RoboDK station: final_robot_station.rdk

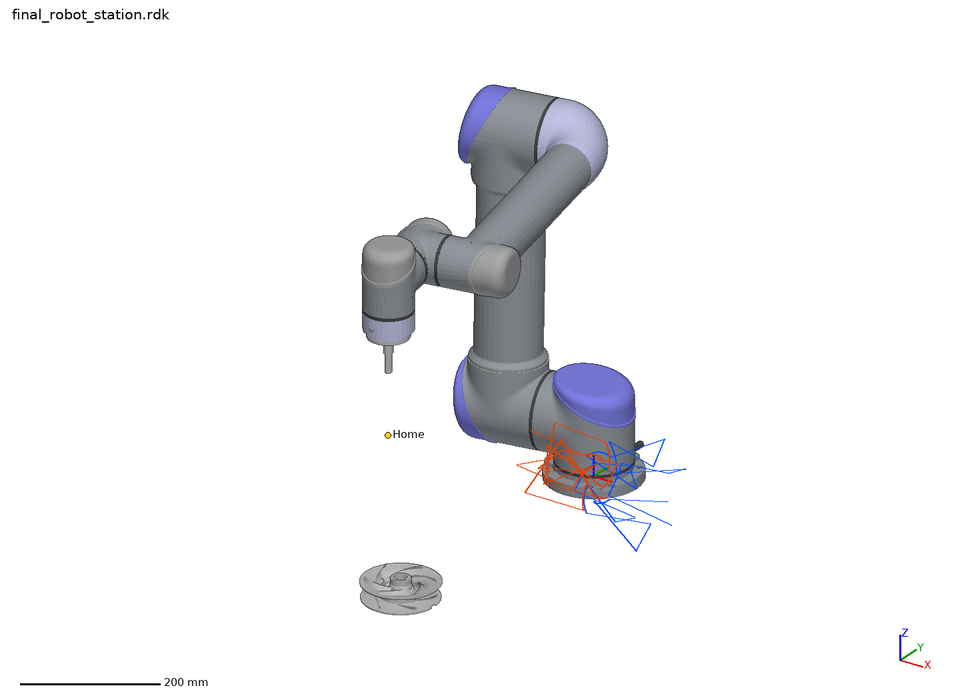
[picture v0: the station drawn from its stored meshes, robots at their saved joint values, targets as dots, program paths as lines]
Station test3. Poses are relative to the parent item; angles as X-Y-Z fixed-axis rotations.
  - frame UR5 Base at (0, 0, 0) mm, rotated rx 0 ry 0 rz -2.6 deg
    - robot UR5: 6 axes, payload 5 kg, reach 850 mm, repeatability 0.1 mm, weight 18.4 kg
        modified DH rows (alpha deg, a mm, theta deg, d mm): 0, 0, 0, 89.2; 90, 0, 180, 0; 0, 425, 0, 0; 0, 392.43, 0, 109; -90, 0, 0, 93.65; 90, 0, 180, 82
        joint limits [-360, -360, -360, -360, -360, -360] to [360, 360, 360, 360, 360, 360]; home [0, -90, -90, 0, 90, 0]; saved at [-76.875, -87.55, -95.198, -87.252, 90, 13.125]
      - tool laser_fixture_tool, TCP at (0, 0, 163) mm, size 63 x 63 x 63 mm
    - target Home (joint target) at (0, -480, 250) mm, rotated rx -180 ry 0 rz -180 deg; joints [-76.875, -87.55, -95.198, -87.252, 90, 13.125] of UR5
  - machining project Path1 settings: rotZ(0) | rotX(0)*rotY(0) | rotz(0) | onStart | onPathStart | onApproach | onPoint | onRetract | onFinish | SetRPM(%1) | SetTool(%1) | Extruder(%1) | default | default | OutOnMov(%1) | OutOffMov(%1) | onPathFinish | M_RunCode(%1)
  - program upper_vane (336 instructions, listed below)
  - machining project Path2 settings: rotZ(0) | rotX(0)*rotY(0) | rotz(0) | onStart | onPathStart | onApproach | onPoint | onRetract | onFinish | SetRPM(%1) | SetTool(%1) | Extruder(%1) | default | default | OutOnMov(%1) | OutOffMov(%1) | onPathFinish | M_RunCode(%1)
  - program lower_vane (305 instructions, listed below)
  - machining project Path3 settings: rotZ(0) | rotX(0)*rotY(0) | rotz(0) | onStart | onPathStart | onApproach | onPoint | onRetract | onFinish | SetRPM(%1) | SetTool(%1) | Extruder(%1) | default | default | OutOnMov(%1) | OutOffMov(%1) | onPathFinish | M_RunCode(%1)
  - program hub (106 instructions, listed below)
  - object PAPER_TEST at (0, -480, 0) mm, size 98 x 86 x 16 mm, geometry from PAPER_TEST.step
  - program MainProgram (19 instructions, listed below)
  - program Path2 (299 instructions, listed below)
  - program Path3 (105 instructions, listed below)
  - frame table at (0, 0, 0) mm
  - object Top_weld_path_dense at (0, -480, 0) mm, rotated rx 0 ry -90 rz 0 deg, size 32.2 x 115.4 x 114.9 mm
  - object Lower_weld_path_dense at (0, 0, 32.2) mm, rotated rx 0 ry 90 rz 0 deg, size 31 x 118.2 x 118.2 mm
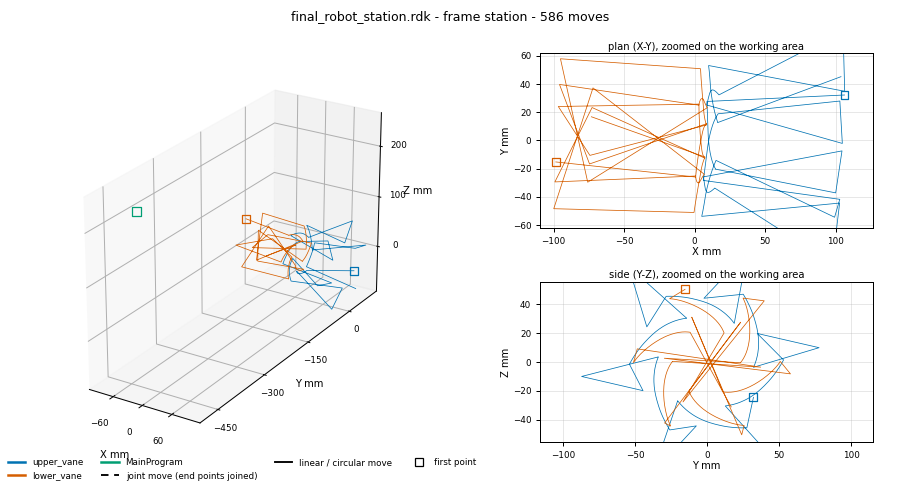
[picture p0: tool path of final_robot_station.rdk in frame station, 586 of 1059 moves have a stored position in this frame; points joined in program order, loops and branches not executed]
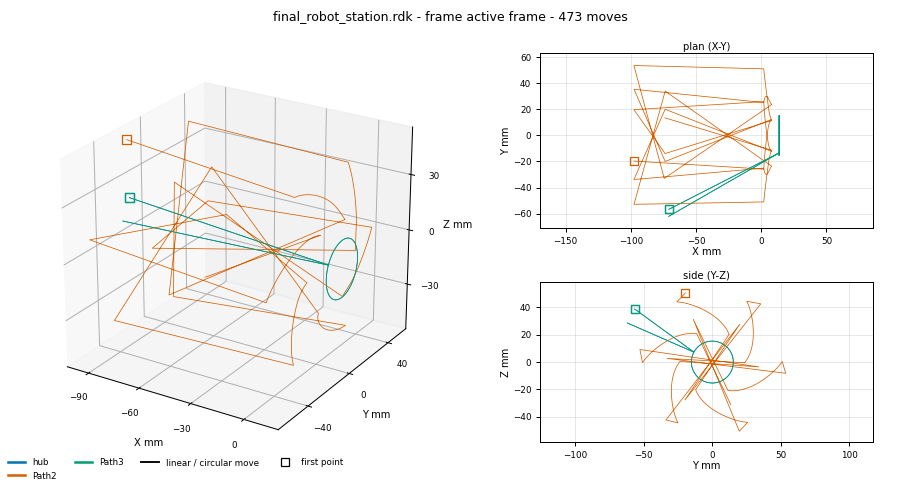
[picture p1: tool path of final_robot_station.rdk in frame active frame, 473 of 1059 moves have a stored position in this frame; points joined in program order, loops and branches not executed]

--- program upper_vane (robot UR5) ---
  Smooth(1)
  Set Ref.: UR5 Base
  Set Tool: laser_fixture_tool
  Show laser_fixture_tool
  Set speed (1000.0 mm/s)
  MoveJ 1 to (104.83, 37.05, -24.45) mm, rotated rx -180 ry -77.76 rz -174.71 deg; joints [-78.761, -85.544, -122.094, -54.774, 100.978, 11.402]
  MoveL 2 to (104.83, 37.05, -24.45) mm, rotated rx -180 ry -77.76 rz -174.71 deg; joints [-78.761, -85.544, -122.094, -54.774, 100.978, 11.402]
  MoveL 3 to (7.52, 28.05, -45.66) mm, rotated rx 180 ry -77.76 rz -174.71 deg; joints [-76.153, -96.353, -128.923, -36.642, 100.622, 14.033]
  MoveL 4 to (7.52, 28.05, -45.66) mm, rotated rx 180 ry -77.76 rz -174.71 deg; joints [-76.153, -96.353, -128.923, -36.642, 100.622, 14.033]
  Set speed (100.0 mm/s)
  Smooth(1)
  MoveL 5 to (7.65, 26.53, -45.69) mm, rotated rx 180 ry -78.61 rz -174.54 deg; joints [-75.694, -96.347, -128.777, -36.756, 99.685, 14.45]
  MoveL 6 to (7.78, 25.01, -45.69) mm, rotated rx -180 ry -79.74 rz -174.38 deg; joints [-75.091, -96.317, -128.596, -37.013, 98.472, 15.003]
  MoveL 7 to (7.91, 23.49, -45.67) mm, rotated rx 180 ry -81.09 rz -174.3 deg; joints [-74.379, -96.291, -128.35, -37.468, 97.046, 15.663]
  MoveL 8 to (8.03, 22.04, -45.61) mm, rotated rx 180 ry -82.56 rz -174.26 deg; joints [-73.616, -96.281, -128.06, -38.061, 95.524, 16.378]
  MoveL 9 to (8.15, 20.65, -45.54) mm, rotated rx 180 ry -84.09 rz -174.26 deg; joints [-72.832, -96.291, -127.75, -38.731, 93.961, 17.121]
  MoveL 10 to (8.26, 19.26, -45.44) mm, rotated rx 180 ry -85.7 rz -174.3 deg; joints [-72.021, -96.337, -127.386, -39.533, 92.34, 17.903]
  MoveL 11 to (8.37, 17.87, -45.32) mm, rotated rx 180 ry -87.36 rz -174.38 deg; joints [-71.197, -96.422, -126.982, -40.43, 90.689, 18.711]
  MoveL 12 to (8.49, 16.49, -45.17) mm, rotated rx 180 ry -89.06 rz -174.48 deg; joints [-70.375, -96.543, -126.553, -41.387, 89.033, 19.533]
  MoveL 13 to (8.6, 15.11, -44.99) mm, rotated rx 0 ry -89.24 rz 5.33 deg; joints [-69.589, -96.729, -126.039, -42.503, 87.434, 20.341]
  MoveL 14 to (8.7, 13.77, -44.79) mm, rotated rx 0 ry -87.62 rz 4.97 deg; joints [-68.892, -96.992, -125.413, -43.811, 85.994, 21.079]
  MoveL 15 to (8.8, 12.48, -44.57) mm, rotated rx 0 ry -86.09 rz 4.54 deg; joints [-68.268, -97.304, -124.741, -45.182, 84.684, 21.758]
  MoveL 16 to (8.9, 11.19, -44.33) mm, rotated rx 0 ry -84.61 rz 3.98 deg; joints [-67.718, -97.686, -123.97, -46.708, 83.499, 22.377]
  MoveL 17 to (9, 9.83, -44.04) mm, rotated rx 0 ry -83.06 rz 3.41 deg; joints [-67.162, -98.115, -123.162, -48.289, 82.283, 23.016]
  MoveL 18 to (9.1, 8.47, -43.73) mm, rotated rx 0 ry -81.52 rz 2.91 deg; joints [-66.609, -98.544, -122.405, -49.771, 81.062, 23.664]
  MoveL 19 to (9.21, 7.11, -43.4) mm, rotated rx 0 ry -79.92 rz 2.67 deg; joints [-65.995, -98.917, -121.82, -50.973, 79.719, 24.393]
  MoveL 20 to (9.32, 5.84, -43.07) mm, rotated rx 0 ry -78.4 rz 2.53 deg; joints [-65.401, -99.258, -121.333, -52.005, 78.412, 25.12]
  MoveL 21 to (9.44, 4.58, -42.73) mm, rotated rx 0 ry -76.9 rz 2.35 deg; joints [-64.845, -99.631, -120.812, -53.094, 77.169, 25.822]
  MoveL 22 to (9.56, 3.42, -42.39) mm, rotated rx 0 ry -75.57 rz 2.15 deg; joints [-64.375, -99.996, -120.31, -54.126, 76.093, 26.437]
  MoveL 23 to (9.67, 2.38, -42.07) mm, rotated rx 0 ry -74.39 rz 2 deg; joints [-63.962, -100.325, -119.878, -55.019, 75.134, 26.993]
  MoveL 24 to (9.79, 1.35, -41.73) mm, rotated rx 0 ry -73.25 rz 1.82 deg; joints [-63.588, -100.667, -119.429, -55.928, 74.241, 27.514]
  MoveL 25 to (9.91, 0.35, -41.38) mm, rotated rx 0 ry -72.21 rz 1.6 deg; joints [-63.268, -101.011, -118.973, -56.827, 73.449, 27.974]
  MoveL 26 to (10.04, -0.61, -41.02) mm, rotated rx 0 ry -71.25 rz 1.39 deg; joints [-62.988, -101.342, -118.538, -57.674, 72.731, 28.39]
  MoveL 27 to (10.18, -1.55, -40.65) mm, rotated rx 0 ry -70.36 rz 1.15 deg; joints [-62.753, -101.677, -118.092, -58.517, 72.092, 28.754]
  MoveL 28 to (10.33, -2.51, -40.24) mm, rotated rx 0 ry -69.54 rz 0.86 deg; joints [-62.564, -102.018, -117.626, -59.366, 71.534, 29.06]
  MoveL 29 to (10.48, -3.45, -39.82) mm, rotated rx 0 ry -68.79 rz 0.57 deg; joints [-62.41, -102.352, -117.166, -60.183, 71.038, 29.32]
  MoveL 30 to (10.65, -4.38, -39.38) mm, rotated rx 0 ry -68.11 rz 0.26 deg; joints [-62.291, -102.677, -116.711, -60.968, 70.604, 29.534]
  MoveL 31 to (10.82, -5.3, -38.92) mm, rotated rx 0 ry -67.47 rz 0 deg; joints [-62.186, -102.982, -116.291, -61.687, 70.191, 29.733]
  MoveL 32 to (11.01, -6.25, -38.41) mm, rotated rx 0 ry -66.89 rz -0.34 deg; joints [-62.125, -103.301, -115.833, -62.437, 69.851, 29.869]
  MoveL 33 to (11.21, -7.19, -37.88) mm, rotated rx 0 ry -66.37 rz -0.67 deg; joints [-62.092, -103.605, -115.389, -63.143, 69.562, 29.964]
  MoveL 34 to (11.42, -8.11, -37.33) mm, rotated rx 0 ry -65.93 rz -1.01 deg; joints [-62.095, -103.898, -114.948, -63.819, 69.339, 30.006]
  MoveL 35 to (11.64, -9.02, -36.76) mm, rotated rx 0 ry -65.54 rz -1.35 deg; joints [-62.117, -104.173, -114.529, -64.444, 69.148, 30.021]
  MoveL 36 to (11.86, -9.91, -36.17) mm, rotated rx 0 ry -65.18 rz -1.65 deg; joints [-62.144, -104.43, -114.137, -65.021, 68.967, 30.026]
  MoveL 37 to (12.1, -10.79, -35.56) mm, rotated rx 0 ry -64.87 rz -1.99 deg; joints [-62.198, -104.685, -113.735, -65.598, 68.834, 29.991]
  MoveL 38 to (12.33, -11.6, -34.96) mm, rotated rx 0 ry -64.54 rz -2.25 deg; joints [-62.224, -104.908, -113.396, -66.098, 68.659, 29.996]
  MoveL 39 to (12.58, -12.39, -34.35) mm, rotated rx 0 ry -64.18 rz -2.48 deg; joints [-62.236, -105.126, -113.072, -66.587, 68.454, 30.023]
  MoveL 40 to (12.84, -13.19, -33.7) mm, rotated rx 0 ry -63.8 rz -2.73 deg; joints [-62.245, -105.354, -112.733, -67.11, 68.233, 30.058]
  MoveL 41 to (13.12, -13.99, -33.01) mm, rotated rx 0 ry -63.4 rz -3.03 deg; joints [-62.261, -105.602, -112.358, -67.695, 68.019, 30.081]
  MoveL 42 to (13.41, -14.77, -32.31) mm, rotated rx 0 ry -62.99 rz -3.38 deg; joints [-62.285, -105.87, -111.95, -68.339, 67.816, 30.092]
  MoveL 43 to (13.7, -15.51, -31.61) mm, rotated rx 0 ry -62.56 rz -3.76 deg; joints [-62.303, -106.15, -111.524, -69.027, 67.609, 30.107]
  MoveL 44 to (14, -16.21, -30.91) mm, rotated rx 0 ry -62.09 rz -4.16 deg; joints [-62.306, -106.443, -111.086, -69.759, 67.376, 30.144]
  MoveL 45 to (14.31, -16.89, -30.2) mm, rotated rx 0 ry -61.58 rz -4.62 deg; joints [-62.308, -106.766, -110.604, -70.575, 67.142, 30.178]
  MoveL 46 to (14.63, -17.55, -29.48) mm, rotated rx 0 ry -61.04 rz -5.16 deg; joints [-62.313, -107.122, -110.072, -71.483, 66.91, 30.203]
  MoveL 47 to (14.97, -18.18, -28.74) mm, rotated rx 0 ry -60.48 rz -5.78 deg; joints [-62.325, -107.517, -109.481, -72.493, 66.694, 30.208]
  MoveL 48 to (15.31, -18.8, -28) mm, rotated rx 0 ry -59.9 rz -6.49 deg; joints [-62.345, -107.949, -108.834, -73.6, 66.494, 30.193]
  MoveL 49 to (15.66, -19.38, -27.25) mm, rotated rx 0 ry -59.71 rz -7.57 deg; joints [-62.575, -108.441, -107.984, -74.851, 66.721, 29.804]
  MoveL 50 to (15.84, -19.66, -26.87) mm, rotated rx 0 ry -60.27 rz -8.58 deg; joints [-63.004, -108.736, -107.315, -75.582, 67.472, 29.074]
  Set speed (1000.0 mm/s)
  MoveL 51 to (15.84, -19.66, -26.87) mm, rotated rx 0 ry -60.27 rz -8.58 deg; joints [-63.004, -108.736, -107.315, -75.582, 67.472, 29.074]
  MoveL 52 to (101.71, -32.61, -76.47) mm, rotated rx 0 ry -60.27 rz -8.58 deg; joints [-59.167, -106.315, -95.895, -90.843, 68.931, 32.896]
  Set speed (1000.0 mm/s)
  MoveL 53 to (104.83, -2.65, -44.31) mm, rotated rx 180 ry -88.39 rz -166.78 deg; joints [-70.24, -87.361, -121.86, -47.778, 87.082, 19.241]
  MoveL 54 to (7.52, -25.52, -47.12) mm, rotated rx -180 ry -88.39 rz -166.78 deg; joints [-70.907, -100.111, -125.994, -30.862, 87.233, 18.59]
  MoveL 55 to (7.52, -25.52, -47.12) mm, rotated rx -180 ry -88.39 rz -166.78 deg; joints [-70.907, -100.111, -125.994, -30.862, 87.233, 18.59]
  Set speed (100.0 mm/s)
  Smooth(1)
  MoveL 56 to (7.65, -26.3, -45.82) mm, rotated rx -180 ry -88.98 rz -167.43 deg; joints [-70.908, -100.255, -125.373, -32.142, 86.887, 18.646]
  MoveL 57 to (7.78, -27.07, -44.51) mm, rotated rx -180 ry -89.68 rz -168.32 deg; joints [-70.892, -100.451, -124.564, -33.83, 86.506, 18.733]
  MoveL 58 to (7.91, -27.8, -43.18) mm, rotated rx 0 ry -89.56 rz 10.56 deg; joints [-70.888, -100.712, -123.582, -35.862, 86.148, 18.82]
  MoveL 59 to (8.03, -28.48, -41.89) mm, rotated rx 0 ry -88.79 rz 9.31 deg; joints [-70.894, -101.028, -122.505, -38.056, 85.822, 18.897]
  MoveL 60 to (8.15, -29.11, -40.65) mm, rotated rx 0 ry -88.01 rz 8 deg; joints [-70.9, -101.391, -121.379, -40.316, 85.512, 18.967]
  MoveL 61 to (8.26, -29.72, -39.4) mm, rotated rx 0 ry -87.24 rz 6.58 deg; joints [-70.926, -101.815, -120.171, -42.69, 85.24, 19.011]
  MoveL 62 to (8.37, -30.31, -38.14) mm, rotated rx 0 ry -86.46 rz 5.1 deg; joints [-70.965, -102.296, -118.908, -45.126, 84.994, 19.032]
  MoveL 63 to (8.49, -30.87, -36.86) mm, rotated rx 0 ry -85.69 rz 3.58 deg; joints [-71.011, -102.824, -117.611, -47.582, 84.761, 19.033]
  MoveL 64 to (8.6, -31.41, -35.58) mm, rotated rx 0 ry -85.01 rz 2.01 deg; joints [-71.107, -103.402, -116.278, -50.039, 84.629, 18.968]
  MoveL 65 to (8.7, -31.91, -34.32) mm, rotated rx 0 ry -84.51 rz 0.42 deg; joints [-71.28, -104.01, -114.951, -52.406, 84.664, 18.804]
  MoveL 66 to (8.8, -32.36, -33.09) mm, rotated rx 0 ry -84.11 rz -1.13 deg; joints [-71.487, -104.628, -113.66, -54.655, 84.776, 18.59]
  MoveL 67 to (8.9, -32.79, -31.86) mm, rotated rx 0 ry -83.86 rz -2.7 deg; joints [-71.756, -105.274, -112.363, -56.851, 85.016, 18.295]
  MoveL 68 to (9, -33.23, -30.53) mm, rotated rx 0 ry -83.59 rz -4.33 deg; joints [-72.028, -105.971, -111.011, -59.116, 85.243, 17.983]
  MoveL 69 to (9.1, -33.64, -29.2) mm, rotated rx 0 ry -83.26 rz -5.93 deg; joints [-72.258, -106.68, -109.682, -61.334, 85.386, 17.703]
  MoveL 70 to (9.21, -34.03, -27.86) mm, rotated rx 0 ry -82.7 rz -7.45 deg; joints [-72.369, -107.39, -108.393, -63.52, 85.284, 17.539]
  MoveL 71 to (9.32, -34.38, -26.6) mm, rotated rx 0 ry -82.07 rz -8.86 deg; joints [-72.426, -108.072, -107.192, -65.559, 85.093, 17.423]
  MoveL 72 to (9.44, -34.72, -25.33) mm, rotated rx 0 ry -81.5 rz -10.27 deg; joints [-72.505, -108.765, -105.998, -67.558, 84.947, 17.275]
  MoveL 73 to (9.56, -35, -24.16) mm, rotated rx 0 ry -81.02 rz -11.54 deg; joints [-72.595, -109.402, -104.922, -69.337, 84.849, 17.114]
  MoveL 74 to (9.67, -35.24, -23.1) mm, rotated rx 0 ry -80.58 rz -12.66 deg; joints [-72.664, -109.975, -103.972, -70.904, 84.735, 16.975]
  MoveL 75 to (9.79, -35.46, -22.03) mm, rotated rx 0 ry -80.19 rz -13.76 deg; joints [-72.748, -110.537, -103.051, -72.407, 84.652, 16.818]
  MoveL 76 to (9.91, -35.66, -21) mm, rotated rx 0 ry -79.87 rz -14.79 deg; joints [-72.849, -111.068, -102.191, -73.796, 84.612, 16.642]
  MoveL 77 to (10.04, -35.83, -19.99) mm, rotated rx 0 ry -79.59 rz -15.75 deg; joints [-72.95, -111.563, -101.397, -75.073, 84.581, 16.468]
  MoveL 78 to (10.18, -35.98, -18.98) mm, rotated rx 0 ry -79.37 rz -16.65 deg; joints [-73.067, -112.032, -100.648, -76.264, 84.584, 16.277]
  MoveL 79 to (10.33, -36.1, -17.95) mm, rotated rx 0 ry -79.22 rz -17.52 deg; joints [-73.206, -112.475, -99.941, -77.374, 84.629, 16.066]
  MoveL 80 to (10.48, -36.21, -16.92) mm, rotated rx 0 ry -79.11 rz -18.32 deg; joints [-73.352, -112.887, -99.286, -78.399, 84.689, 15.851]
  MoveL 81 to (10.65, -36.29, -15.9) mm, rotated rx 0 ry -79.04 rz -19.07 deg; joints [-73.505, -113.268, -98.68, -79.34, 84.765, 15.633]
  MoveL 82 to (10.82, -36.35, -14.87) mm, rotated rx 0 ry -78.96 rz -19.76 deg; joints [-73.646, -113.621, -98.121, -80.216, 84.818, 15.431]
  MoveL 83 to (11.01, -36.39, -13.79) mm, rotated rx 0 ry -78.95 rz -20.43 deg; joints [-73.816, -113.954, -97.588, -81.037, 84.922, 15.201]
  MoveL 84 to (11.21, -36.4, -12.71) mm, rotated rx 0 ry -78.98 rz -21.04 deg; joints [-73.99, -114.253, -97.108, -81.777, 85.035, 14.974]
  MoveL 85 to (11.42, -36.39, -11.64) mm, rotated rx 0 ry -79.05 rz -21.59 deg; joints [-74.174, -114.516, -96.681, -82.431, 85.17, 14.743]
  MoveL 86 to (11.64, -36.35, -10.57) mm, rotated rx 0 ry -79.14 rz -22.09 deg; joints [-74.355, -114.747, -96.3, -83.018, 85.301, 14.521]
  MoveL 87 to (11.86, -36.28, -9.5) mm, rotated rx 0 ry -79.21 rz -22.55 deg; joints [-74.526, -114.958, -95.951, -83.564, 85.414, 14.312]
  MoveL 88 to (12.1, -36.19, -8.44) mm, rotated rx 0 ry -79.33 rz -22.97 deg; joints [-74.71, -115.147, -95.632, -84.06, 85.556, 14.095]
  MoveL 89 to (12.33, -36.07, -7.44) mm, rotated rx 0 ry -79.38 rz -23.38 deg; joints [-74.857, -115.328, -95.329, -84.549, 85.639, 13.914]
  MoveL 90 to (12.58, -35.94, -6.44) mm, rotated rx 0 ry -79.4 rz -23.8 deg; joints [-74.992, -115.517, -95.017, -85.06, 85.697, 13.745]
  MoveL 91 to (12.84, -35.78, -5.43) mm, rotated rx 0 ry -79.41 rz -24.25 deg; joints [-75.129, -115.719, -94.686, -85.609, 85.758, 13.57]
  MoveL 92 to (13.12, -35.58, -4.39) mm, rotated rx 0 ry -79.46 rz -24.74 deg; joints [-75.282, -115.935, -94.331, -86.192, 85.846, 13.377]
  MoveL 93 to (13.41, -35.36, -3.36) mm, rotated rx 0 ry -79.54 rz -25.25 deg; joints [-75.449, -116.165, -93.956, -86.804, 85.967, 13.168]
  MoveL 94 to (13.7, -35.13, -2.37) mm, rotated rx 0 ry -79.63 rz -25.8 deg; joints [-75.617, -116.412, -93.558, -87.45, 86.101, 12.953]
  MoveL 95 to (14, -34.88, -1.42) mm, rotated rx 0 ry -79.72 rz -26.4 deg; joints [-75.783, -116.685, -93.124, -88.153, 86.237, 12.737]
  MoveL 96 to (14.31, -34.6, -0.47) mm, rotated rx 0 ry -79.83 rz -27.05 deg; joints [-75.962, -116.989, -92.649, -88.915, 86.404, 12.502]
  MoveL 97 to (14.63, -34.3, 0.46) mm, rotated rx 0 ry -79.98 rz -27.76 deg; joints [-76.157, -117.324, -92.13, -89.74, 86.607, 12.246]
  MoveL 98 to (14.97, -33.98, 1.38) mm, rotated rx 0 ry -80.19 rz -28.52 deg; joints [-76.373, -117.689, -91.568, -90.622, 86.858, 11.965]
  MoveL 99 to (15.31, -33.64, 2.28) mm, rotated rx 0 ry -80.44 rz -29.34 deg; joints [-76.61, -118.086, -90.964, -91.559, 87.154, 11.661]
  MoveL 100 to (15.66, -33.29, 3.16) mm, rotated rx 0 ry -81.17 rz -29.97 deg; joints [-77.008, -118.36, -90.513, -92.187, 87.784, 11.239]
  MoveL 101 to (15.84, -33.1, 3.59) mm, rotated rx 0 ry -82.19 rz -29.93 deg; joints [-77.434, -118.27, -90.576, -91.96, 88.565, 10.872]
  Set speed (1000.0 mm/s)
  MoveL 102 to (15.84, -33.1, 3.59) mm, rotated rx 0 ry -82.19 rz -29.93 deg; joints [-77.434, -118.27, -90.576, -91.96, 88.565, 10.872]
  MoveL 103 to (101.71, -82.53, -9.99) mm, rotated rx 0 ry -82.19 rz -29.93 deg; joints [-77.222, -120.426, -73.678, -106.707, 88.674, 11.054]
  Set speed (1000.0 mm/s)
  MoveL 104 to (104.83, -39.7, -19.86) mm, rotated rx 0 ry -79.4 rz 8.11 deg; joints [-69.534, -94.529, -112.106, -59.512, 77.242, 20.788]
  MoveL 105 to (7.52, -53.56, -1.46) mm, rotated rx 0 ry -79.4 rz 8.11 deg; joints [-72.132, -104.254, -117.716, -43.595, 77.429, 18.133]
  MoveL 106 to (7.52, -53.56, -1.46) mm, rotated rx 0 ry -79.4 rz 8.11 deg; joints [-72.132, -104.254, -117.716, -43.595, 77.429, 18.133]
  Set speed (100.0 mm/s)
  Smooth(1)
  MoveL 107 to (7.65, -52.83, -0.13) mm, rotated rx 0 ry -79.66 rz 7.26 deg; joints [-72.499, -104.351, -117.217, -44.647, 77.958, 17.76]
  MoveL 108 to (7.78, -52.08, 1.19) mm, rotated rx 0 ry -80.07 rz 6.18 deg; joints [-72.964, -104.514, -116.551, -45.96, 78.697, 17.279]
  MoveL 109 to (7.91, -51.29, 2.49) mm, rotated rx 0 ry -80.65 rz 4.94 deg; joints [-73.523, -104.733, -115.763, -47.441, 79.637, 16.694]
  MoveL 110 to (8.03, -50.52, 3.72) mm, rotated rx 0 ry -81.34 rz 3.63 deg; joints [-74.127, -104.996, -114.914, -48.986, 80.68, 16.058]
  MoveL 111 to (8.15, -49.76, 4.89) mm, rotated rx 0 ry -82.08 rz 2.28 deg; joints [-74.746, -105.3, -114.026, -50.568, 81.764, 15.405]
  MoveL 112 to (8.26, -48.98, 6.04) mm, rotated rx 0 ry -82.92 rz 0.89 deg; joints [-75.4, -105.642, -113.098, -52.188, 82.924, 14.712]
  MoveL 113 to (8.37, -48.18, 7.18) mm, rotated rx 0 ry -83.82 rz -0.52 deg; joints [-76.075, -106.021, -112.143, -53.836, 84.125, 14]
  MoveL 114 to (8.49, -47.36, 8.3) mm, rotated rx 0 ry -84.75 rz -1.95 deg; joints [-76.753, -106.433, -111.169, -55.502, 85.336, 13.284]
  MoveL 115 to (8.6, -46.52, 9.41) mm, rotated rx 0 ry -85.77 rz -3.33 deg; joints [-77.454, -106.851, -110.233, -57.081, 86.594, 12.547]
  MoveL 116 to (8.7, -45.68, 10.47) mm, rotated rx 0 ry -86.89 rz -4.55 deg; joints [-78.169, -107.237, -109.409, -58.442, 87.889, 11.802]
  MoveL 117 to (8.8, -44.84, 11.48) mm, rotated rx 0 ry -88.03 rz -5.66 deg; joints [-78.868, -107.604, -108.665, -59.666, 89.16, 11.078]
  MoveL 118 to (8.9, -43.98, 12.47) mm, rotated rx 0 ry -89.26 rz -6.66 deg; joints [-79.587, -107.944, -108.008, -60.734, 90.474, 10.342]
  MoveL 119 to (9, -43.06, 13.51) mm, rotated rx 180 ry -89.47 rz 172.29 deg; joints [-80.323, -108.318, -107.317, -61.878, 91.816, 9.593]
  MoveL 120 to (9.1, -42.11, 14.53) mm, rotated rx 180 ry -88.27 rz 171.2 deg; joints [-81.021, -108.726, -106.593, -63.107, 93.079, 8.885]
  MoveL 121 to (9.21, -41.14, 15.54) mm, rotated rx 180 ry -87.26 rz 169.94 deg; joints [-81.635, -109.218, -105.728, -64.612, 94.169, 8.257]
  MoveL 122 to (9.32, -40.22, 16.48) mm, rotated rx 180 ry -86.38 rz 168.69 deg; joints [-82.175, -109.727, -104.856, -66.144, 95.115, 7.703]
  MoveL 123 to (9.44, -39.29, 17.4) mm, rotated rx -180 ry -85.49 rz 167.47 deg; joints [-82.71, -110.229, -104.021, -67.616, 96.055, 7.156]
  MoveL 124 to (9.56, -38.42, 18.23) mm, rotated rx 180 ry -84.66 rz 166.41 deg; joints [-83.192, -110.678, -103.295, -68.904, 96.903, 6.665]
  MoveL 125 to (9.67, -37.62, 18.97) mm, rotated rx 180 ry -83.95 rz 165.45 deg; joints [-83.606, -111.09, -102.638, -70.081, 97.623, 6.244]
  MoveL 126 to (9.79, -36.81, 19.7) mm, rotated rx 180 ry -83.24 rz 164.54 deg; joints [-84.009, -111.481, -102.027, -71.187, 98.325, 5.835]
  MoveL 127 to (9.91, -36.01, 20.38) mm, rotated rx 180 ry -82.55 rz 163.72 deg; joints [-84.392, -111.833, -101.49, -72.175, 98.991, 5.45]
  MoveL 128 to (10.04, -35.22, 21.04) mm, rotated rx 180 ry -81.9 rz 162.97 deg; joints [-84.745, -112.155, -101.006, -73.082, 99.602, 5.095]
  MoveL 129 to (10.18, -34.42, 21.67) mm, rotated rx 180 ry -81.27 rz 162.3 deg; joints [-85.086, -112.441, -100.585, -73.894, 100.19, 4.756]
  MoveL 130 to (10.33, -33.6, 22.29) mm, rotated rx 180 ry -80.64 rz 161.7 deg; joints [-85.419, -112.688, -100.231, -74.605, 100.765, 4.427]
  MoveL 131 to (10.48, -32.76, 22.9) mm, rotated rx 180 ry -80.05 rz 161.17 deg; joints [-85.735, -112.903, -99.93, -75.241, 101.305, 4.117]
  MoveL 132 to (10.65, -31.91, 23.48) mm, rotated rx -180 ry -79.47 rz 160.69 deg; joints [-86.034, -113.085, -99.679, -75.801, 101.815, 3.824]
  MoveL 133 to (10.82, -31.05, 24.05) mm, rotated rx -180 ry -78.95 rz 160.24 deg; joints [-86.308, -113.253, -99.448, -76.34, 102.277, 3.556]
  MoveL 134 to (11.01, -30.14, 24.62) mm, rotated rx 180 ry -78.41 rz 159.86 deg; joints [-86.588, -113.378, -99.285, -76.782, 102.747, 3.285]
  MoveL 135 to (11.21, -29.21, 25.17) mm, rotated rx -180 ry -77.9 rz 159.54 deg; joints [-86.849, -113.471, -99.17, -77.154, 103.185, 3.032]
  MoveL 136 to (11.42, -28.27, 25.69) mm, rotated rx 180 ry -77.41 rz 159.29 deg; joints [-87.097, -113.525, -99.113, -77.437, 103.598, 2.793]
  MoveL 137 to (11.64, -27.32, 26.19) mm, rotated rx -180 ry -76.97 rz 159.08 deg; joints [-87.327, -113.555, -99.089, -77.675, 103.976, 2.573]
  MoveL 138 to (11.86, -26.37, 26.67) mm, rotated rx 180 ry -76.55 rz 158.88 deg; joints [-87.539, -113.575, -99.075, -77.902, 104.324, 2.369]
  MoveL 139 to (12.1, -25.4, 27.12) mm, rotated rx 180 ry -76.14 rz 158.73 deg; joints [-87.748, -113.565, -99.105, -78.061, 104.668, 2.17]
  MoveL 140 to (12.33, -24.48, 27.52) mm, rotated rx 180 ry -75.78 rz 158.54 deg; joints [-87.93, -113.582, -99.091, -78.285, 104.967, 1.994]
  MoveL 141 to (12.58, -23.55, 27.9) mm, rotated rx -180 ry -75.43 rz 158.31 deg; joints [-88.107, -113.614, -99.051, -78.556, 105.259, 1.823]
  MoveL 142 to (12.84, -22.59, 28.27) mm, rotated rx -180 ry -75.06 rz 158.06 deg; joints [-88.292, -113.654, -99, -78.852, 105.571, 1.645]
  MoveL 143 to (13.12, -21.59, 28.62) mm, rotated rx 180 ry -74.64 rz 157.81 deg; joints [-88.493, -113.692, -98.959, -79.143, 105.919, 1.451]
  MoveL 144 to (13.41, -20.59, 28.95) mm, rotated rx 180 ry -74.18 rz 157.58 deg; joints [-88.709, -113.729, -98.927, -79.423, 106.305, 1.243]
  MoveL 145 to (13.7, -19.62, 29.24) mm, rotated rx -180 ry -73.69 rz 157.33 deg; joints [-88.934, -113.778, -98.884, -79.718, 106.716, 1.027]
  MoveL 146 to (14, -18.66, 29.49) mm, rotated rx 180 ry -73.17 rz 157.04 deg; joints [-89.168, -113.852, -98.811, -80.059, 107.155, 0.802]
  MoveL 147 to (14.31, -17.71, 29.73) mm, rotated rx 180 ry -72.58 rz 156.75 deg; joints [-89.423, -113.937, -98.733, -80.416, 107.644, 0.556]
  MoveL 148 to (14.63, -16.76, 29.94) mm, rotated rx 180 ry -71.93 rz 156.44 deg; joints [-89.702, -114.034, -98.651, -80.783, 108.189, 0.288]
  MoveL 149 to (14.97, -15.8, 30.12) mm, rotated rx -180 ry -71.2 rz 156.14 deg; joints [-90.007, -114.136, -98.577, -81.146, 108.796, -0.006]
  MoveL 150 to (15.31, -14.85, 30.28) mm, rotated rx -180 ry -70.4 rz 155.85 deg; joints [-90.336, -114.245, -98.51, -81.505, 109.462, -0.326]
  MoveL 151 to (15.66, -13.91, 30.41) mm, rotated rx -180 ry -69.47 rz 156.07 deg; joints [-90.715, -114.109, -98.833, -81.229, 110.241, -0.697]
  MoveL 152 to (15.84, -13.44, 30.46) mm, rotated rx 180 ry -68.89 rz 156.98 deg; joints [-90.952, -113.656, -99.593, -80.102, 110.734, -0.937]
  Set speed (1000.0 mm/s)
  MoveL 153 to (15.84, -13.44, 30.46) mm, rotated rx 180 ry -68.89 rz 156.98 deg; joints [-90.952, -113.656, -99.593, -80.102, 110.734, -0.937]
  MoveL 154 to (101.71, -49.91, 66.48) mm, rotated rx -180 ry -68.89 rz 156.98 deg; joints [-94.194, -113.921, -84.944, -95.571, 109.42, -4.093]
  Set speed (1000.0 mm/s)
  MoveL 155 to (104.83, -37.05, 24.45) mm, rotated rx 0 ry -77.76 rz -5.29 deg; joints [-75.431, -100.004, -102.645, -75.565, 79.48, 14.759]
  MoveL 156 to (7.52, -28.05, 45.66) mm, rotated rx 0 ry -77.76 rz -5.29 deg; joints [-77.455, -105.732, -111.895, -60.21, 79.198, 12.72]
  MoveL 157 to (7.52, -28.05, 45.66) mm, rotated rx 0 ry -77.76 rz -5.29 deg; joints [-77.455, -105.732, -111.895, -60.21, 79.198, 12.72]
  Set speed (100.0 mm/s)
  Smooth(1)
  MoveL 158 to (7.65, -26.53, 45.69) mm, rotated rx 0 ry -78.61 rz -5.46 deg; joints [-77.828, -105.583, -111.973, -60.197, 80.02, 12.305]
  MoveL 159 to (7.78, -25.01, 45.69) mm, rotated rx 0 ry -79.74 rz -5.62 deg; joints [-78.323, -105.425, -112.063, -60.097, 81.088, 11.764]
  MoveL 160 to (7.91, -23.49, 45.67) mm, rotated rx 0 ry -81.09 rz -5.7 deg; joints [-78.917, -105.245, -112.195, -59.871, 82.354, 11.127]
  MoveL 161 to (8.03, -22.04, 45.61) mm, rotated rx 0 ry -82.56 rz -5.74 deg; joints [-79.564, -105.065, -112.352, -59.57, 83.72, 10.447]
  MoveL 162 to (8.15, -20.65, 45.54) mm, rotated rx 0 ry -84.09 rz -5.74 deg; joints [-80.241, -104.901, -112.513, -59.246, 85.142, 9.745]
  MoveL 163 to (8.26, -19.26, 45.44) mm, rotated rx 0 ry -85.7 rz -5.7 deg; joints [-80.957, -104.735, -112.707, -58.86, 86.643, 9.013]
  MoveL 164 to (8.37, -17.87, 45.32) mm, rotated rx 0 ry -87.36 rz -5.62 deg; joints [-81.702, -104.578, -112.921, -58.44, 88.2, 8.262]
  MoveL 165 to (8.49, -16.49, 45.17) mm, rotated rx 0 ry -89.06 rz -5.52 deg; joints [-82.464, -104.438, -113.141, -58.018, 89.792, 7.501]
  MoveL 166 to (8.6, -15.11, 44.99) mm, rotated rx 180 ry -89.24 rz 174.67 deg; joints [-83.224, -104.281, -113.434, -57.484, 91.381, 6.749]
  MoveL 167 to (8.7, -13.77, 44.79) mm, rotated rx 180 ry -87.62 rz 175.03 deg; joints [-83.941, -104.082, -113.842, -56.768, 92.888, 6.043]
  MoveL 168 to (8.8, -12.48, 44.57) mm, rotated rx 180 ry -86.09 rz 175.46 deg; joints [-84.621, -103.878, -114.296, -55.984, 94.321, 5.377]
  MoveL 169 to (8.9, -11.19, 44.33) mm, rotated rx 180 ry -84.61 rz 176.02 deg; joints [-85.274, -103.639, -114.849, -55.038, 95.704, 4.738]
  MoveL 170 to (9, -9.83, 44.04) mm, rotated rx 180 ry -83.06 rz 176.59 deg; joints [-85.959, -103.418, -115.414, -54.08, 97.163, 4.066]
  MoveL 171 to (9.1, -8.47, 43.73) mm, rotated rx -180 ry -81.52 rz 177.09 deg; joints [-86.65, -103.252, -115.911, -53.247, 98.639, 3.384]
  MoveL 172 to (9.21, -7.11, 43.4) mm, rotated rx 180 ry -79.92 rz 177.33 deg; joints [-87.376, -103.21, -116.21, -52.777, 100.189, 2.664]
  MoveL 173 to (9.32, -5.84, 43.07) mm, rotated rx 180 ry -78.4 rz 177.47 deg; joints [-88.072, -103.23, -116.409, -52.496, 101.68, 1.967]
  MoveL 174 to (9.44, -4.58, 42.73) mm, rotated rx -180 ry -76.9 rz 177.65 deg; joints [-88.75, -103.248, -116.638, -52.173, 103.144, 1.282]
  MoveL 175 to (9.56, -3.42, 42.39) mm, rotated rx 180 ry -75.57 rz 177.85 deg; joints [-89.351, -103.263, -116.872, -51.847, 104.45, 0.67]
  MoveL 176 to (9.67, -2.38, 42.07) mm, rotated rx 180 ry -74.39 rz 178 deg; joints [-89.884, -103.297, -117.059, -51.611, 105.617, 0.12]
  MoveL 177 to (9.79, -1.35, 41.73) mm, rotated rx 180 ry -73.25 rz 178.18 deg; joints [-90.39, -103.322, -117.266, -51.346, 106.736, -0.407]
  MoveL 178 to (9.91, -0.35, 41.38) mm, rotated rx -180 ry -72.21 rz 178.4 deg; joints [-90.851, -103.333, -117.497, -51.044, 107.766, -0.893]
  MoveL 179 to (10.04, 0.61, 41.02) mm, rotated rx 180 ry -71.25 rz 178.61 deg; joints [-91.271, -103.342, -117.721, -50.759, 108.717, -1.342]
  MoveL 180 to (10.18, 1.55, 40.65) mm, rotated rx -180 ry -70.36 rz 178.85 deg; joints [-91.655, -103.334, -117.971, -50.434, 109.601, -1.756]
  MoveL 181 to (10.33, 2.51, 40.24) mm, rotated rx -180 ry -69.54 rz 179.14 deg; joints [-92.003, -103.302, -118.254, -50.053, 110.417, -2.137]
  MoveL 182 to (10.48, 3.45, 39.82) mm, rotated rx -180 ry -68.79 rz 179.43 deg; joints [-92.316, -103.26, -118.546, -49.662, 111.169, -2.484]
  MoveL 183 to (10.65, 4.38, 39.38) mm, rotated rx 180 ry -68.11 rz 179.74 deg; joints [-92.596, -103.205, -118.847, -49.256, 111.856, -2.798]
  MoveL 184 to (10.82, 5.3, 38.92) mm, rotated rx 180 ry -67.47 rz -180 deg; joints [-92.854, -103.155, -119.124, -48.899, 112.502, -3.089]
  MoveL 185 to (11.01, 6.25, 38.41) mm, rotated rx -180 ry -66.89 rz -179.66 deg; joints [-93.08, -103.072, -119.453, -48.454, 113.095, -3.349]
  MoveL 186 to (11.21, 7.19, 37.88) mm, rotated rx -180 ry -66.37 rz -179.33 deg; joints [-93.274, -102.977, -119.784, -48.004, 113.625, -3.574]
  MoveL 187 to (11.42, 8.11, 37.33) mm, rotated rx 180 ry -65.93 rz -178.99 deg; joints [-93.431, -102.864, -120.13, -47.526, 114.083, -3.758]
  MoveL 188 to (11.64, 9.02, 36.76) mm, rotated rx 180 ry -65.54 rz -178.65 deg; joints [-93.561, -102.744, -120.467, -47.064, 114.492, -3.913]
  MoveL 189 to (11.86, 9.91, 36.17) mm, rotated rx -180 ry -65.18 rz -178.35 deg; joints [-93.676, -102.628, -120.785, -46.636, 114.872, -4.051]
  MoveL 190 to (12.1, 10.79, 35.56) mm, rotated rx 180 ry -64.87 rz -178.01 deg; joints [-93.766, -102.495, -121.124, -46.164, 115.207, -4.161]
  MoveL 191 to (12.33, 11.6, 34.96) mm, rotated rx 180 ry -64.54 rz -177.75 deg; joints [-93.863, -102.395, -121.399, -45.804, 115.553, -4.28]
  MoveL 192 to (12.58, 12.39, 34.35) mm, rotated rx 180 ry -64.18 rz -177.52 deg; joints [-93.97, -102.311, -121.651, -45.482, 115.924, -4.411]
  MoveL 193 to (12.84, 13.19, 33.7) mm, rotated rx 180 ry -63.8 rz -177.27 deg; joints [-94.086, -102.231, -121.912, -45.143, 116.325, -4.554]
  MoveL 194 to (13.12, 13.99, 33.01) mm, rotated rx -180 ry -63.4 rz -176.97 deg; joints [-94.206, -102.143, -122.204, -44.736, 116.745, -4.704]
  MoveL 195 to (13.41, 14.77, 32.31) mm, rotated rx -180 ry -62.99 rz -176.62 deg; joints [-94.33, -102.052, -122.524, -44.26, 117.18, -4.86]
  MoveL 196 to (13.7, 15.51, 31.61) mm, rotated rx -180 ry -62.56 rz -176.24 deg; joints [-94.466, -101.969, -122.852, -43.746, 117.64, -5.032]
  MoveL 197 to (14, 16.21, 30.91) mm, rotated rx 180 ry -62.09 rz -175.84 deg; joints [-94.624, -101.906, -123.18, -43.214, 118.147, -5.232]
  MoveL 198 to (14.31, 16.89, 30.2) mm, rotated rx -180 ry -61.58 rz -175.38 deg; joints [-94.798, -101.847, -123.538, -42.602, 118.695, -5.454]
  MoveL 199 to (14.63, 17.55, 29.48) mm, rotated rx -180 ry -61.04 rz -174.84 deg; joints [-94.988, -101.793, -123.933, -41.892, 119.285, -5.698]
  MoveL 200 to (14.97, 18.18, 28.74) mm, rotated rx 180 ry -60.48 rz -174.22 deg; joints [-95.191, -101.742, -124.373, -41.062, 119.908, -5.961]
  MoveL 201 to (15.31, 18.8, 28) mm, rotated rx 180 ry -59.9 rz -173.51 deg; joints [-95.407, -101.697, -124.857, -40.111, 120.565, -6.242]
  MoveL 202 to (15.66, 19.38, 27.25) mm, rotated rx -180 ry -59.71 rz -172.43 deg; joints [-95.453, -101.478, -125.618, -38.535, 120.854, -6.3]
  MoveL 203 to (15.84, 19.66, 26.87) mm, rotated rx 180 ry -60.27 rz -171.42 deg; joints [-95.19, -101.095, -126.372, -36.938, 120.374, -5.951]
  Set speed (1000.0 mm/s)
  MoveL 204 to (15.84, 19.66, 26.87) mm, rotated rx 180 ry -60.27 rz -171.42 deg; joints [-95.19, -101.095, -126.372, -36.938, 120.374, -5.951]
  MoveL 205 to (101.71, 32.61, 76.47) mm, rotated rx 180 ry -60.27 rz -171.42 deg; joints [-101.773, -92.531, -118.876, -56.886, 120.794, -13.584]
  Set speed (1000.0 mm/s)
  MoveL 206 to (104.83, 2.65, 44.31) mm, rotated rx 0 ry -88.39 rz -13.22 deg; joints [-82.252, -99.108, -102.424, -81.785, 90.173, 7.541]
  MoveL 207 to (7.52, 25.52, 47.12) mm, rotated rx 0 ry -88.39 rz -13.22 deg; joints [-82.218, -102.992, -113.944, -66.381, 90.181, 7.575]
  MoveL 208 to (7.52, 25.52, 47.12) mm, rotated rx 0 ry -88.39 rz -13.22 deg; joints [-82.218, -102.992, -113.944, -66.381, 90.181, 7.575]
  Set speed (100.0 mm/s)
  Smooth(1)
  MoveL 209 to (7.65, 26.3, 45.82) mm, rotated rx 0 ry -88.98 rz -12.57 deg; joints [-82.3, -102.584, -114.537, -65.477, 90.656, 7.514]
  MoveL 210 to (7.78, 27.07, 44.51) mm, rotated rx 0 ry -89.68 rz -11.68 deg; joints [-82.425, -102.071, -115.307, -64.243, 91.209, 7.419]
  MoveL 211 to (7.91, 27.8, 43.18) mm, rotated rx 180 ry -89.56 rz 169.44 deg; joints [-82.564, -101.468, -116.241, -62.704, 91.792, 7.313]
  MoveL 212 to (8.03, 28.48, 41.89) mm, rotated rx 180 ry -88.79 rz 170.69 deg; joints [-82.71, -100.83, -117.261, -60.991, 92.375, 7.2]
  MoveL 213 to (8.15, 29.11, 40.65) mm, rotated rx 180 ry -88.01 rz 172 deg; joints [-82.865, -100.191, -118.318, -59.18, 92.962, 7.074]
  MoveL 214 to (8.26, 29.72, 39.4) mm, rotated rx 180 ry -87.24 rz 173.42 deg; joints [-83.015, -99.533, -119.446, -57.22, 93.542, 6.952]
  MoveL 215 to (8.37, 30.31, 38.14) mm, rotated rx 180 ry -86.46 rz 174.9 deg; joints [-83.162, -98.875, -120.62, -55.15, 94.118, 6.828]
  MoveL 216 to (8.49, 30.87, 36.86) mm, rotated rx 180 ry -85.69 rz 176.42 deg; joints [-83.309, -98.235, -121.814, -53.006, 94.696, 6.7]
  MoveL 217 to (8.6, 31.41, 35.58) mm, rotated rx 180 ry -85.01 rz 177.99 deg; joints [-83.407, -97.601, -123.044, -50.776, 95.188, 6.616]
  MoveL 218 to (8.7, 31.91, 34.32) mm, rotated rx -180 ry -84.51 rz 179.58 deg; joints [-83.413, -96.983, -124.281, -48.525, 95.504, 6.618]
  MoveL 219 to (8.8, 32.36, 33.09) mm, rotated rx 180 ry -84.11 rz -178.87 deg; joints [-83.365, -96.405, -125.485, -46.308, 95.717, 6.667]
  MoveL 220 to (8.9, 32.79, 31.86) mm, rotated rx 180 ry -83.86 rz -177.3 deg; joints [-83.231, -95.839, -126.703, -44.053, 95.777, 6.796]
  MoveL 221 to (9, 33.23, 30.53) mm, rotated rx 180 ry -83.59 rz -175.67 deg; joints [-83.087, -95.29, -127.962, -41.673, 95.837, 6.929]
  MoveL 222 to (9.1, 33.64, 29.2) mm, rotated rx -180 ry -83.26 rz -174.07 deg; joints [-82.978, -94.806, -129.179, -39.306, 95.962, 7.023]
  MoveL 223 to (9.21, 34.03, 27.86) mm, rotated rx 180 ry -82.7 rz -172.55 deg; joints [-83.012, -94.425, -130.319, -36.974, 96.347, 6.972]
  MoveL 224 to (9.32, 34.38, 26.6) mm, rotated rx 180 ry -82.07 rz -171.14 deg; joints [-83.103, -94.134, -131.357, -34.768, 96.818, 6.863]
  MoveL 225 to (9.44, 34.72, 25.33) mm, rotated rx 180 ry -81.5 rz -169.73 deg; joints [-83.162, -93.877, -132.386, -32.541, 97.23, 6.782]
  MoveL 226 to (9.56, 35, 24.16) mm, rotated rx -180 ry -81.02 rz -168.46 deg; joints [-83.186, -93.677, -133.31, -30.504, 97.555, 6.734]
  MoveL 227 to (9.67, 35.24, 23.1) mm, rotated rx 180 ry -80.58 rz -167.34 deg; joints [-83.22, -93.537, -134.115, -28.678, 97.872, 6.677]
  MoveL 228 to (9.79, 35.46, 22.03) mm, rotated rx 180 ry -80.19 rz -166.24 deg; joints [-83.225, -93.423, -134.895, -26.884, 98.137, 6.647]
  MoveL 229 to (9.91, 35.66, 21) mm, rotated rx 180 ry -79.87 rz -165.21 deg; joints [-83.191, -93.331, -135.624, -25.185, 98.325, 6.653]
  MoveL 230 to (10.04, 35.83, 19.99) mm, rotated rx 180 ry -79.59 rz -164.25 deg; joints [-83.145, -93.267, -136.294, -23.596, 98.482, 6.67]
  MoveL 231 to (10.18, 35.98, 18.98) mm, rotated rx 180 ry -79.37 rz -163.35 deg; joints [-83.06, -93.215, -136.928, -22.081, 98.571, 6.723]
  MoveL 232 to (10.33, 36.1, 17.95) mm, rotated rx 180 ry -79.22 rz -162.48 deg; joints [-82.93, -93.169, -137.53, -20.637, 98.58, 6.817]
  MoveL 233 to (10.48, 36.21, 16.92) mm, rotated rx -180 ry -79.11 rz -161.68 deg; joints [-82.776, -93.135, -138.089, -19.283, 98.546, 6.933]
  MoveL 234 to (10.65, 36.29, 15.9) mm, rotated rx 180 ry -79.04 rz -160.93 deg; joints [-82.598, -93.107, -138.608, -18.02, 98.467, 7.071]
  MoveL 235 to (10.82, 36.35, 14.87) mm, rotated rx 180 ry -78.96 rz -160.24 deg; joints [-82.427, -93.096, -139.083, -16.838, 98.402, 7.202]
  MoveL 236 to (11.01, 36.39, 13.79) mm, rotated rx 180 ry -78.95 rz -159.57 deg; joints [-82.197, -93.076, -139.543, -15.709, 98.239, 7.386]
  MoveL 237 to (11.21, 36.4, 12.71) mm, rotated rx 180 ry -78.98 rz -158.96 deg; joints [-81.948, -93.057, -139.959, -14.683, 98.043, 7.587]
  MoveL 238 to (11.42, 36.39, 11.64) mm, rotated rx 180 ry -79.05 rz -158.41 deg; joints [-81.67, -93.031, -140.335, -13.769, 97.792, 7.814]
  MoveL 239 to (11.64, 36.35, 10.57) mm, rotated rx -180 ry -79.14 rz -157.91 deg; joints [-81.387, -93.007, -140.671, -12.947, 97.531, 8.047]
  MoveL 240 to (11.86, 36.28, 9.5) mm, rotated rx 180 ry -79.21 rz -157.45 deg; joints [-81.113, -92.99, -140.977, -12.187, 97.284, 8.271]
  MoveL 241 to (12.1, 36.19, 8.44) mm, rotated rx -180 ry -79.33 rz -157.03 deg; joints [-80.808, -92.963, -141.26, -11.495, 96.98, 8.521]
  MoveL 242 to (12.33, 36.07, 7.44) mm, rotated rx 180 ry -79.38 rz -156.62 deg; joints [-80.564, -92.961, -141.519, -10.819, 96.77, 8.716]
  MoveL 243 to (12.58, 35.94, 6.44) mm, rotated rx 180 ry -79.4 rz -156.2 deg; joints [-80.342, -92.976, -141.778, -10.113, 96.596, 8.89]
  MoveL 244 to (12.84, 35.78, 5.43) mm, rotated rx 180 ry -79.41 rz -155.75 deg; joints [-80.111, -93.001, -142.05, -9.353, 96.412, 9.066]
  MoveL 245 to (13.12, 35.58, 4.39) mm, rotated rx -180 ry -79.46 rz -155.26 deg; joints [-79.85, -93.03, -142.341, -8.541, 96.176, 9.264]
  MoveL 246 to (13.41, 35.36, 3.36) mm, rotated rx 180 ry -79.54 rz -154.75 deg; joints [-79.56, -93.062, -142.648, -7.684, 95.885, 9.483]
  MoveL 247 to (13.7, 35.13, 2.37) mm, rotated rx 180 ry -79.63 rz -154.2 deg; joints [-79.261, -93.106, -142.971, -6.771, 95.57, 9.703]
  MoveL 248 to (14, 34.88, 1.42) mm, rotated rx 180 ry -79.72 rz -153.6 deg; joints [-78.967, -93.174, -143.317, -5.769, 95.251, 9.913]
  MoveL 249 to (14.31, 34.6, 0.47) mm, rotated rx 180 ry -79.83 rz -152.95 deg; joints [-78.642, -93.257, -143.694, -4.671, 94.874, 10.139]
  MoveL 250 to (14.63, 34.3, -0.46) mm, rotated rx 180 ry -79.98 rz -152.24 deg; joints [-78.279, -93.358, -144.103, -3.472, 94.427, 10.387]
  MoveL 251 to (14.97, 33.98, -1.38) mm, rotated rx 180 ry -80.19 rz -151.48 deg; joints [-77.867, -93.476, -144.545, -2.179, 93.886, 10.667]
  MoveL 252 to (15.31, 33.64, -2.28) mm, rotated rx 180 ry -80.44 rz -150.66 deg; joints [-77.405, -93.615, -145.018, -0.794, 93.251, 10.975]
  MoveL 253 to (15.66, 33.29, -3.16) mm, rotated rx -180 ry -81.17 rz -150.03 deg; joints [-76.605, -93.576, -145.41, 0.059, 92.008, 11.584]
  MoveL 254 to (15.84, 33.1, -3.59) mm, rotated rx 180 ry -82.19 rz -150.07 deg; joints [-75.744, -93.257, -145.439, -0.472, 90.569, 12.323]
  Set speed (1000.0 mm/s)
  MoveL 255 to (15.84, 33.1, -3.59) mm, rotated rx 180 ry -82.19 rz -150.07 deg; joints [-75.744, -93.257, -145.439, -0.472, 90.569, 12.323]
  MoveL 256 to (101.71, 82.53, 9.99) mm, rotated rx 180 ry -82.19 rz -150.07 deg; joints [-75.965, -70.134, -144.82, -24.216, 90.682, 12.133]
  Set speed (1000.0 mm/s)
  MoveL 257 to (104.83, 39.7, 19.86) mm, rotated rx 180 ry -79.4 rz 171.89 deg; joints [-84.634, -91.952, -111.978, -73.147, 101.312, 5.417]
  MoveL 258 to (7.52, 53.56, 1.46) mm, rotated rx -180 ry -79.4 rz 171.89 deg; joints [-82.148, -97.744, -122.527, -56.305, 101.607, 7.937]
  MoveL 259 to (7.52, 53.56, 1.46) mm, rotated rx -180 ry -79.4 rz 171.89 deg; joints [-82.148, -97.744, -122.527, -56.305, 101.607, 7.937]
  Set speed (100.0 mm/s)
  Smooth(1)
  MoveL 260 to (7.65, 52.83, 0.13) mm, rotated rx -180 ry -79.66 rz 172.74 deg; joints [-81.792, -97.412, -123.04, -55.248, 101.272, 8.303]
  MoveL 261 to (7.78, 52.08, -1.19) mm, rotated rx -180 ry -80.07 rz 173.82 deg; joints [-81.334, -96.976, -123.71, -53.919, 100.749, 8.771]
  MoveL 262 to (7.91, 51.29, -2.49) mm, rotated rx 180 ry -80.65 rz 175.06 deg; joints [-80.761, -96.466, -124.493, -52.406, 100.02, 9.348]
  MoveL 263 to (8.03, 50.52, -3.72) mm, rotated rx 180 ry -81.34 rz 176.37 deg; joints [-80.12, -95.931, -125.325, -50.823, 99.153, 9.988]
  MoveL 264 to (8.15, 49.76, -4.89) mm, rotated rx 180 ry -82.08 rz 177.72 deg; joints [-79.438, -95.394, -126.181, -49.21, 98.2, 10.664]
  MoveL 265 to (8.26, 48.98, -6.04) mm, rotated rx 180 ry -82.92 rz 179.11 deg; joints [-78.685, -94.854, -127.063, -47.564, 97.118, 11.402]
  MoveL 266 to (8.37, 48.18, -7.18) mm, rotated rx -180 ry -83.82 rz -179.48 deg; joints [-77.877, -94.324, -127.957, -45.906, 95.935, 12.189]
  MoveL 267 to (8.49, 47.36, -8.3) mm, rotated rx 180 ry -84.75 rz -178.05 deg; joints [-77.03, -93.815, -128.854, -44.249, 94.679, 13.007]
  MoveL 268 to (8.6, 46.52, -9.41) mm, rotated rx -180 ry -85.77 rz -176.67 deg; joints [-76.119, -93.347, -129.702, -42.707, 93.308, 13.881]
  MoveL 269 to (8.7, 45.68, -10.47) mm, rotated rx 180 ry -86.89 rz -175.45 deg; joints [-75.159, -92.95, -130.431, -41.427, 91.842, 14.801]
  MoveL 270 to (8.8, 44.84, -11.48) mm, rotated rx -180 ry -88.03 rz -174.34 deg; joints [-74.194, -92.613, -131.073, -40.33, 90.354, 15.728]
  MoveL 271 to (8.9, 43.98, -12.47) mm, rotated rx 180 ry -89.26 rz -173.34 deg; joints [-73.185, -92.335, -131.618, -39.455, 88.785, 16.702]
  MoveL 272 to (9, 43.06, -13.51) mm, rotated rx 0 ry -89.47 rz 7.71 deg; joints [-72.126, -92.079, -132.175, -38.565, 87.134, 17.73]
  MoveL 273 to (9.1, 42.11, -14.53) mm, rotated rx 0 ry -88.27 rz 8.8 deg; joints [-71.093, -91.85, -132.748, -37.628, 85.519, 18.735]
  MoveL 274 to (9.21, 41.14, -15.54) mm, rotated rx 0 ry -87.26 rz 10.06 deg; joints [-70.13, -91.616, -133.442, -36.396, 84.015, 19.664]
  MoveL 275 to (9.32, 40.22, -16.48) mm, rotated rx 0 ry -86.38 rz 11.31 deg; joints [-69.242, -91.414, -134.141, -35.118, 82.624, 20.513]
  MoveL 276 to (9.44, 39.29, -17.4) mm, rotated rx 0 ry -85.49 rz 12.53 deg; joints [-68.343, -91.256, -134.792, -33.934, 81.203, 21.38]
  MoveL 277 to (9.56, 38.42, -18.23) mm, rotated rx 0 ry -84.66 rz 13.59 deg; joints [-67.52, -91.15, -135.343, -32.94, 79.893, 22.18]
  MoveL 278 to (9.67, 37.62, -18.97) mm, rotated rx 0 ry -83.95 rz 14.55 deg; joints [-66.794, -91.078, -135.835, -32.03, 78.732, 22.885]
  MoveL 279 to (9.79, 36.81, -19.7) mm, rotated rx 0 ry -83.24 rz 15.46 deg; joints [-66.082, -91.038, -136.279, -31.21, 77.584, 23.586]
  MoveL 280 to (9.91, 36.01, -20.38) mm, rotated rx 0 ry -82.55 rz 16.28 deg; joints [-65.407, -91.028, -136.653, -30.525, 76.489, 24.259]
  MoveL 281 to (10.04, 35.22, -21.04) mm, rotated rx 0 ry -81.9 rz 17.03 deg; joints [-64.781, -91.042, -136.98, -29.917, 75.467, 24.89]
  MoveL 282 to (10.18, 34.42, -21.67) mm, rotated rx 0 ry -81.27 rz 17.7 deg; joints [-64.185, -91.08, -137.246, -29.422, 74.486, 25.502]
  MoveL 283 to (10.33, 33.6, -22.29) mm, rotated rx 0 ry -80.64 rz 18.3 deg; joints [-63.616, -91.141, -137.448, -29.051, 73.544, 26.1]
  MoveL 284 to (10.48, 32.76, -22.9) mm, rotated rx 0 ry -80.05 rz 18.83 deg; joints [-63.086, -91.218, -137.603, -28.761, 72.659, 26.668]
  MoveL 285 to (10.65, 31.91, -23.48) mm, rotated rx 0 ry -79.47 rz 19.31 deg; joints [-62.595, -91.309, -137.712, -28.551, 71.831, 27.206]
  MoveL 286 to (10.82, 31.05, -24.05) mm, rotated rx 0 ry -78.95 rz 19.76 deg; joints [-62.145, -91.407, -137.807, -28.342, 71.065, 27.702]
  MoveL 287 to (11.01, 30.14, -24.62) mm, rotated rx 0 ry -78.41 rz 20.14 deg; joints [-61.713, -91.524, -137.834, -28.269, 70.321, 28.198]
  MoveL 288 to (11.21, 29.21, -25.17) mm, rotated rx 0 ry -77.9 rz 20.46 deg; joints [-61.323, -91.648, -137.821, -28.26, 69.64, 28.657]
  MoveL 289 to (11.42, 28.27, -25.69) mm, rotated rx 0 ry -77.41 rz 20.71 deg; joints [-60.975, -91.78, -137.758, -28.342, 69.023, 29.082]
  MoveL 290 to (11.64, 27.32, -26.19) mm, rotated rx 0 ry -76.97 rz 20.92 deg; joints [-60.667, -91.915, -137.67, -28.455, 68.467, 29.467]
  MoveL 291 to (11.86, 26.37, -26.67) mm, rotated rx 0 ry -76.55 rz 21.12 deg; joints [-60.389, -92.049, -137.576, -28.56, 67.954, 29.82]
  MoveL 292 to (12.1, 25.4, -27.12) mm, rotated rx 0 ry -76.14 rz 21.27 deg; joints [-60.134, -92.189, -137.442, -28.748, 67.474, 30.158]
  MoveL 293 to (12.33, 24.48, -27.52) mm, rotated rx 0 ry -75.78 rz 21.46 deg; joints [-59.901, -92.316, -137.356, -28.822, 67.024, 30.461]
  MoveL 294 to (12.58, 23.55, -27.9) mm, rotated rx 0 ry -75.43 rz 21.69 deg; joints [-59.666, -92.441, -137.294, -28.842, 66.564, 30.762]
  MoveL 295 to (12.84, 22.59, -28.27) mm, rotated rx 0 ry -75.06 rz 21.94 deg; joints [-59.42, -92.572, -137.234, -28.859, 66.072, 31.083]
  MoveL 296 to (13.12, 21.59, -28.62) mm, rotated rx 0 ry -74.64 rz 22.19 deg; joints [-59.158, -92.713, -137.156, -28.925, 65.541, 31.434]
  MoveL 297 to (13.41, 20.59, -28.95) mm, rotated rx 0 ry -74.18 rz 22.42 deg; joints [-58.883, -92.861, -137.061, -29.048, 64.976, 31.816]
  MoveL 298 to (13.7, 19.62, -29.24) mm, rotated rx 0 ry -73.69 rz 22.67 deg; joints [-58.595, -93.012, -136.969, -29.188, 64.378, 32.226]
  MoveL 299 to (14, 18.66, -29.49) mm, rotated rx 0 ry -73.17 rz 22.96 deg; joints [-58.285, -93.165, -136.896, -29.312, 63.731, 32.671]
  MoveL 300 to (14.31, 17.71, -29.73) mm, rotated rx 0 ry -72.58 rz 23.25 deg; joints [-57.948, -93.329, -136.815, -29.485, 63.025, 33.168]
  MoveL 301 to (14.63, 16.76, -29.94) mm, rotated rx 0 ry -71.93 rz 23.56 deg; joints [-57.584, -93.506, -136.721, -29.721, 62.256, 33.725]
  MoveL 302 to (14.97, 15.8, -30.12) mm, rotated rx 0 ry -71.2 rz 23.86 deg; joints [-57.195, -93.699, -136.601, -30.049, 61.426, 34.347]
  MoveL 303 to (15.31, 14.85, -30.28) mm, rotated rx 0 ry -70.4 rz 24.15 deg; joints [-56.783, -93.908, -136.457, -30.47, 60.542, 35.036]
  MoveL 304 to (15.66, 13.91, -30.41) mm, rotated rx 0 ry -69.47 rz 23.93 deg; joints [-56.481, -94.153, -135.939, -31.732, 59.857, 35.709]
  MoveL 305 to (15.84, 13.44, -30.46) mm, rotated rx 0 ry -68.89 rz 23.02 deg; joints [-56.531, -94.329, -135.129, -33.526, 59.895, 35.924]
  Set speed (1000.0 mm/s)
  MoveL 306 to (15.84, 13.44, -30.46) mm, rotated rx 0 ry -68.89 rz 23.02 deg; joints [-56.531, -94.329, -135.129, -33.526, 59.895, 35.924]
  MoveL 307 to (101.71, 49.91, -66.48) mm, rotated rx 0 ry -68.89 rz 23.02 deg; joints [-48.643, -80.047, -130.531, -57.031, 59.247, 45.044]
  Smooth(1)

--- program lower_vane (robot UR5) ---
  Smooth(1)
  Set Ref.: UR5 Base
  Set Tool: laser_fixture_tool
  Show laser_fixture_tool
  Set speed (1000.0 mm/s)
  MoveJ 1 to (-97.68, -19.69, 50.49) mm, rotated rx 180 ry 86.28 rz 176.44 deg; joints [-69.317, -92.399, -109.007, -66.579, 85.26, 20.715]
  MoveL 2 to (-97.68, -19.69, 50.49) mm, rotated rx 180 ry 86.28 rz 176.44 deg; joints [-69.317, -92.399, -109.007, -66.579, 85.26, 20.715]
  MoveL 3 to (1.91, -25.89, 44) mm, rotated rx 180 ry 86.28 rz 176.44 deg; joints [-70.301, -100.232, -116.842, -50.831, 85.295, 19.728]
  MoveL 4 to (1.91, -25.89, 44) mm, rotated rx 180 ry 86.28 rz 176.44 deg; joints [-70.301, -100.232, -116.842, -50.831, 85.295, 19.728]
  Set speed (100.0 mm/s)
  Smooth(1)
  MoveL 5 to (1.98, -24.59, 43.9) mm, rotated rx -180 ry 86.86 rz 176.07 deg; joints [-70.477, -99.929, -117.389, -50.025, 85.726, 19.532]
  MoveL 6 to (2.06, -23.31, 43.74) mm, rotated rx -180 ry 87.81 rz 175.89 deg; joints [-70.872, -99.694, -117.818, -49.325, 86.585, 19.112]
  MoveL 7 to (2.12, -22.3, 43.59) mm, rotated rx -180 ry 88.79 rz 175.78 deg; joints [-71.308, -99.524, -118.156, -48.711, 87.5, 18.658]
  MoveL 8 to (2.19, -21.29, 43.41) mm, rotated rx 180 ry 89.93 rz 175.76 deg; joints [-71.846, -99.394, -118.44, -48.154, 88.61, 18.108]
  MoveL 9 to (2.26, -20.27, 43.2) mm, rotated rx 0 ry 88.78 rz -4.17 deg; joints [-72.484, -99.314, -118.658, -47.684, 89.913, 17.468]
  MoveL 10 to (2.33, -19.25, 42.96) mm, rotated rx 0 ry 87.38 rz -4 deg; joints [-73.195, -99.285, -118.808, -47.321, 91.353, 16.768]
  MoveL 11 to (2.41, -18.24, 42.7) mm, rotated rx 0 ry 85.9 rz -3.77 deg; joints [-73.961, -99.303, -118.906, -47.041, 92.898, 16.024]
  MoveL 12 to (2.5, -17.15, 42.4) mm, rotated rx 0 ry 84.25 rz -3.43 deg; joints [-74.836, -99.379, -118.944, -46.865, 94.654, 15.187]
  MoveL 13 to (2.6, -15.98, 42.05) mm, rotated rx 0 ry 82.45 rz -2.96 deg; joints [-75.804, -99.526, -118.902, -46.846, 96.593, 14.273]
  MoveL 14 to (2.71, -14.82, 41.67) mm, rotated rx 0 ry 80.66 rz -2.39 deg; joints [-76.777, -99.737, -118.774, -47.01, 98.539, 13.363]
  MoveL 15 to (2.81, -13.7, 41.29) mm, rotated rx 0 ry 78.96 rz -1.77 deg; joints [-77.71, -99.991, -118.589, -47.313, 100.405, 12.493]
  MoveL 16 to (2.92, -12.62, 40.89) mm, rotated rx 0 ry 77.35 rz -1.12 deg; joints [-78.593, -100.274, -118.364, -47.727, 102.17, 11.671]
  MoveL 17 to (3.02, -11.55, 40.47) mm, rotated rx 0 ry 75.79 rz -0.41 deg; joints [-79.452, -100.591, -118.095, -48.254, 103.888, 10.869]
  MoveL 18 to (3.14, -10.42, 40.01) mm, rotated rx 0 ry 74.19 rz 0.42 deg; joints [-80.332, -100.971, -117.738, -48.984, 105.647, 10.044]
  MoveL 19 to (3.26, -9.3, 39.53) mm, rotated rx 0 ry 72.65 rz 1.33 deg; joints [-81.18, -101.389, -117.325, -49.857, 107.343, 9.241]
  MoveL 20 to (3.38, -8.19, 39.02) mm, rotated rx 0 ry 71.17 rz 2.33 deg; joints [-81.991, -101.846, -116.845, -50.896, 108.966, 8.465]
  MoveL 21 to (3.5, -7.16, 38.53) mm, rotated rx 0 ry 69.83 rz 3.32 deg; joints [-82.72, -102.299, -116.359, -51.968, 110.422, 7.758]
  MoveL 22 to (3.62, -6.13, 38.01) mm, rotated rx 0 ry 68.57 rz 4.35 deg; joints [-83.403, -102.767, -115.841, -53.132, 111.782, 7.086]
  MoveL 23 to (3.74, -5.11, 37.48) mm, rotated rx 0 ry 67.41 rz 5.41 deg; joints [-84.03, -103.24, -115.299, -54.369, 113.025, 6.459]
  MoveL 24 to (3.87, -4.1, 36.93) mm, rotated rx 0 ry 66.37 rz 6.49 deg; joints [-84.595, -103.709, -114.743, -55.658, 114.132, 5.886]
  MoveL 25 to (3.99, -3.1, 36.36) mm, rotated rx 0 ry 65.46 rz 7.57 deg; joints [-85.091, -104.162, -114.185, -56.968, 115.088, 5.374]
  MoveL 26 to (4.12, -2.14, 35.78) mm, rotated rx 0 ry 64.71 rz 8.61 deg; joints [-85.512, -104.582, -113.65, -58.242, 115.88, 4.933]
  MoveL 27 to (4.25, -1.18, 35.18) mm, rotated rx 0 ry 64.11 rz 9.64 deg; joints [-85.861, -104.982, -113.106, -59.537, 116.51, 4.561]
  MoveL 28 to (4.37, -0.31, 34.6) mm, rotated rx 0 ry 63.69 rz 10.57 deg; joints [-86.126, -105.328, -112.61, -60.72, 116.96, 4.273]
  MoveL 29 to (4.5, 0.55, 34.01) mm, rotated rx 0 ry 63.41 rz 11.52 deg; joints [-86.33, -105.661, -112.097, -61.931, 117.269, 4.046]
  MoveL 30 to (4.62, 1.39, 33.4) mm, rotated rx 0 ry 63.28 rz 12.49 deg; joints [-86.471, -105.983, -111.558, -63.179, 117.433, 3.883]
  MoveL 31 to (4.74, 2.19, 32.8) mm, rotated rx 0 ry 63.13 rz 13.23 deg; joints [-86.612, -106.23, -111.169, -64.129, 117.599, 3.722]
  MoveL 32 to (4.91, 3.31, 31.9) mm, rotated rx 0 ry 63.31 rz 14.51 deg; joints [-86.657, -106.619, -110.427, -65.803, 117.479, 3.648]
  MoveL 33 to (5.08, 4.4, 30.96) mm, rotated rx 0 ry 63.73 rz 15.74 deg; joints [-86.608, -106.972, -109.688, -67.433, 117.142, 3.669]
  MoveL 34 to (5.25, 5.45, 29.99) mm, rotated rx 0 ry 64.15 rz 16.71 deg; joints [-86.559, -107.234, -109.124, -68.717, 116.797, 3.692]
  MoveL 35 to (5.43, 6.44, 28.99) mm, rotated rx 0 ry 64.46 rz 17.42 deg; joints [-86.546, -107.413, -108.742, -69.65, 116.523, 3.684]
  MoveL 36 to (5.61, 7.35, 28) mm, rotated rx 0 ry 64.65 rz 17.92 deg; joints [-86.582, -107.533, -108.502, -70.306, 116.358, 3.63]
  MoveL 37 to (5.8, 8.16, 27.05) mm, rotated rx 0 ry 64.66 rz 18.26 deg; joints [-86.682, -107.618, -108.377, -70.736, 116.338, 3.516]
  MoveL 38 to (6.01, 8.91, 26.1) mm, rotated rx 0 ry 64.51 rz 18.53 deg; joints [-86.845, -107.699, -108.311, -71.052, 116.453, 3.341]
  MoveL 39 to (6.25, 9.59, 25.16) mm, rotated rx 0 ry 64.22 rz 18.78 deg; joints [-87.066, -107.804, -108.258, -71.338, 116.691, 3.11]
  MoveL 40 to (6.49, 10.19, 24.25) mm, rotated rx 0 ry 63.76 rz 19.03 deg; joints [-87.352, -107.943, -108.208, -71.613, 117.077, 2.812]
  MoveL 41 to (6.77, 10.75, 23.33) mm, rotated rx 0 ry 63.16 rz 19.35 deg; joints [-87.697, -108.146, -108.112, -71.974, 117.585, 2.452]
  MoveL 42 to (7.09, 11.26, 22.39) mm, rotated rx 0 ry 62.44 rz 19.8 deg; joints [-88.089, -108.426, -107.94, -72.477, 118.191, 2.04]
  MoveL 43 to (7.44, 11.72, 21.44) mm, rotated rx 0 ry 61.65 rz 20.38 deg; joints [-88.509, -108.792, -107.671, -73.155, 118.859, 1.596]
  MoveL 44 to (7.81, 12.11, 20.53) mm, rotated rx 0 ry 61.24 rz 21.2 deg; joints [-88.775, -109.217, -107.205, -74.142, 119.197, 1.309]
  MoveL 45 to (7.95, 12.23, 20.22) mm, rotated rx 0 ry 61.39 rz 21.56 deg; joints [-88.75, -109.361, -106.959, -74.599, 119.061, 1.33]
  Set speed (1000.0 mm/s)
  MoveL 46 to (7.95, 12.23, 20.22) mm, rotated rx 0 ry 61.39 rz 21.56 deg; joints [-88.75, -109.361, -106.959, -74.599, 119.061, 1.33]
  MoveL 47 to (-73.7, -20.03, -27.66) mm, rotated rx 0 ry 61.39 rz 21.56 deg; joints [-93.535, -108.888, -93.322, -91.083, 117.259, -3.698]
  Set speed (1000.0 mm/s)
  MoveL 48 to (-97.55, 35.36, 42.52) mm, rotated rx 0 ry 88.91 rz -5.86 deg; joints [-69.853, -83.267, -118.799, -62.061, 89.01, 20.041]
  MoveL 49 to (1.91, 25.16, 44.42) mm, rotated rx 0 ry 88.91 rz -5.86 deg; joints [-70.09, -92.894, -126.543, -44.686, 89.035, 19.805]
  MoveL 50 to (1.91, 25.16, 44.42) mm, rotated rx 0 ry 88.91 rz -5.86 deg; joints [-70.09, -92.894, -126.543, -44.686, 89.035, 19.805]
  Set speed (100.0 mm/s)
  Smooth(1)
  MoveL 51 to (1.98, 25.72, 43.25) mm, rotated rx 0 ry 88.27 rz -5.54 deg; joints [-70.632, -92.939, -126.472, -44.789, 89.8, 19.274]
  MoveL 52 to (2.06, 26.23, 42.05) mm, rotated rx 0 ry 87.66 rz -4.79 deg; joints [-71.242, -93.145, -126.069, -45.498, 90.678, 18.692]
  MoveL 53 to (2.12, 26.6, 41.1) mm, rotated rx 0 ry 87.05 rz -4 deg; joints [-71.831, -93.395, -125.614, -46.267, 91.56, 18.13]
  MoveL 54 to (2.19, 26.95, 40.14) mm, rotated rx 0 ry 86.42 rz -3.03 deg; joints [-72.453, -93.726, -125.018, -47.284, 92.499, 17.539]
  MoveL 55 to (2.26, 27.27, 39.15) mm, rotated rx 0 ry 85.81 rz -1.88 deg; joints [-73.092, -94.143, -124.276, -48.567, 93.462, 16.93]
  MoveL 56 to (2.33, 27.58, 38.15) mm, rotated rx 0 ry 85.24 rz -0.58 deg; joints [-73.724, -94.63, -123.425, -50.052, 94.408, 16.324]
  MoveL 57 to (2.41, 27.86, 37.15) mm, rotated rx 0 ry 84.67 rz 0.82 deg; joints [-74.357, -95.179, -122.493, -51.674, 95.353, 15.712]
  MoveL 58 to (2.5, 28.14, 36.05) mm, rotated rx 0 ry 84.1 rz 2.42 deg; joints [-75.015, -95.835, -121.407, -53.568, 96.326, 15.065]
  MoveL 59 to (2.6, 28.42, 34.87) mm, rotated rx 0 ry 83.57 rz 4.22 deg; joints [-75.672, -96.597, -120.174, -55.724, 97.276, 14.407]
  MoveL 60 to (2.71, 28.68, 33.67) mm, rotated rx 0 ry 83.15 rz 6.07 deg; joints [-76.259, -97.403, -118.896, -57.963, 98.097, 13.803]
  MoveL 61 to (2.81, 28.9, 32.51) mm, rotated rx 0 ry 82.81 rz 7.86 deg; joints [-76.775, -98.215, -117.639, -60.159, 98.792, 13.257]
  MoveL 62 to (2.92, 29.1, 31.38) mm, rotated rx 0 ry 82.54 rz 9.59 deg; joints [-77.233, -99.018, -116.423, -62.274, 99.388, 12.759]
  MoveL 63 to (3.02, 29.28, 30.24) mm, rotated rx 0 ry 82.31 rz 11.3 deg; joints [-77.657, -99.837, -115.213, -64.368, 99.917, 12.286]
  MoveL 64 to (3.14, 29.44, 29.03) mm, rotated rx 0 ry 82.19 rz 13.11 deg; joints [-78.032, -100.719, -113.923, -66.597, 100.34, 11.846]
  MoveL 65 to (3.26, 29.58, 27.82) mm, rotated rx 0 ry 82.15 rz 14.91 deg; joints [-78.358, -101.615, -112.635, -68.811, 100.669, 11.445]
  MoveL 66 to (3.38, 29.7, 26.61) mm, rotated rx 0 ry 82.23 rz 16.69 deg; joints [-78.618, -102.522, -111.346, -71.017, 100.873, 11.099]
  MoveL 67 to (3.5, 29.79, 25.46) mm, rotated rx 0 ry 82.34 rz 18.33 deg; joints [-78.836, -103.379, -110.149, -73.049, 101.015, 10.792]
  MoveL 68 to (3.62, 29.86, 24.31) mm, rotated rx 0 ry 82.52 rz 19.93 deg; joints [-79.016, -104.225, -108.984, -75.016, 101.083, 10.518]
  MoveL 69 to (3.74, 29.91, 23.17) mm, rotated rx 0 ry 82.75 rz 21.45 deg; joints [-79.156, -105.045, -107.868, -76.891, 101.077, 10.279]
  MoveL 70 to (3.87, 29.93, 22.02) mm, rotated rx 0 ry 83.05 rz 22.87 deg; joints [-79.257, -105.825, -106.817, -78.648, 100.996, 10.077]
  MoveL 71 to (3.99, 29.93, 20.87) mm, rotated rx 0 ry 83.42 rz 24.16 deg; joints [-79.317, -106.549, -105.848, -80.261, 100.84, 9.916]
  MoveL 72 to (4.12, 29.91, 19.74) mm, rotated rx 0 ry 83.79 rz 25.31 deg; joints [-79.359, -107.201, -104.985, -81.688, 100.652, 9.78]
  MoveL 73 to (4.25, 29.87, 18.61) mm, rotated rx 0 ry 84.26 rz 26.32 deg; joints [-79.347, -107.783, -104.214, -82.965, 100.365, 9.697]
  MoveL 74 to (4.37, 29.81, 17.57) mm, rotated rx 0 ry 84.67 rz 27.15 deg; joints [-79.335, -108.266, -103.58, -84.006, 100.097, 9.629]
  MoveL 75 to (4.5, 29.73, 16.53) mm, rotated rx 0 ry 85.17 rz 27.86 deg; joints [-79.279, -108.689, -103.021, -84.927, 99.749, 9.606]
  MoveL 76 to (4.62, 29.62, 15.5) mm, rotated rx 0 ry 85.79 rz 28.45 deg; joints [-79.163, -109.048, -102.538, -85.727, 99.287, 9.643]
  MoveL 77 to (4.74, 29.5, 14.5) mm, rotated rx 0 ry 85.83 rz 29.04 deg; joints [-79.29, -109.412, -102.095, -86.415, 99.285, 9.476]
  MoveL 78 to (4.91, 29.28, 13.09) mm, rotated rx 0 ry 86.77 rz 29.56 deg; joints [-79.075, -109.754, -101.626, -87.196, 98.551, 9.596]
  MoveL 79 to (5.08, 29.01, 11.67) mm, rotated rx 0 ry 87.98 rz 29.85 deg; joints [-78.726, -109.963, -101.314, -87.743, 97.571, 9.849]
  MoveL 80 to (5.25, 28.69, 10.28) mm, rotated rx 0 ry 89.05 rz 30 deg; joints [-78.428, -110.104, -101.105, -88.117, 96.688, 10.074]
  MoveL 81 to (5.43, 28.33, 8.92) mm, rotated rx 0 ry 89.88 rz 30.1 deg; joints [-78.224, -110.22, -100.945, -88.385, 95.987, 10.226]
  MoveL 82 to (5.61, 27.93, 7.64) mm, rotated rx -180 ry 89.52 rz -149.8 deg; joints [-78.114, -110.341, -100.791, -88.613, 95.472, 10.302]
  MoveL 83 to (5.8, 27.51, 6.46) mm, rotated rx -180 ry 89.18 rz -149.64 deg; joints [-78.11, -110.505, -100.598, -88.87, 95.173, 10.282]
  MoveL 84 to (6.01, 27.06, 5.34) mm, rotated rx -180 ry 89.01 rz -149.37 deg; joints [-78.177, -110.727, -100.34, -89.2, 95.017, 10.194]
  MoveL 85 to (6.25, 26.58, 4.28) mm, rotated rx -180 ry 88.93 rz -149.01 deg; joints [-78.284, -111.014, -100.008, -89.627, 94.945, 10.062]
  MoveL 86 to (6.49, 26.1, 3.3) mm, rotated rx 180 ry 88.99 rz -148.49 deg; joints [-78.454, -111.398, -99.564, -90.207, 95.007, 9.863]
  MoveL 87 to (6.77, 25.58, 2.36) mm, rotated rx 180 ry 89.08 rz -147.81 deg; joints [-78.645, -111.882, -99.004, -90.955, 95.114, 9.63]
  MoveL 88 to (7.09, 25.02, 1.44) mm, rotated rx 180 ry 89.16 rz -146.98 deg; joints [-78.835, -112.464, -98.33, -91.871, 95.226, 9.382]
  MoveL 89 to (7.44, 24.43, 0.58) mm, rotated rx 180 ry 89.19 rz -146.01 deg; joints [-79.007, -113.132, -97.557, -92.937, 95.315, 9.137]
  MoveL 90 to (7.81, 23.83, -0.22) mm, rotated rx -180 ry 88.7 rz -145.38 deg; joints [-78.936, -113.608, -97.009, -93.705, 94.974, 9.121]
  MoveL 91 to (7.95, 23.62, -0.48) mm, rotated rx -180 ry 88.19 rz -145.47 deg; joints [-78.751, -113.593, -97.031, -93.681, 94.565, 9.278]
  Set speed (1000.0 mm/s)
  MoveL 92 to (7.95, 23.62, -0.48) mm, rotated rx 180 ry 88.19 rz -145.47 deg; joints [-78.751, -113.593, -97.031, -93.681, 94.565, 9.278]
  MoveL 93 to (-74.39, -33.03, 2.67) mm, rotated rx -180 ry 88.19 rz -145.47 deg; joints [-79.461, -116.318, -79.804, -108.228, 94.164, 8.689]
  Set speed (1000.0 mm/s)
  MoveL 94 to (-97.68, 53.58, -8.19) mm, rotated rx 0 ry 85.06 rz -1.45 deg; joints [-78.992, -82.845, -118.192, -66.592, 94.573, 11.04]
  MoveL 95 to (1.91, 51.05, 0.42) mm, rotated rx 0 ry 85.06 rz -1.45 deg; joints [-77.878, -91.073, -127.344, -49.123, 94.526, 12.157]
  MoveL 96 to (1.91, 51.05, 0.42) mm, rotated rx 0 ry 85.06 rz -1.45 deg; joints [-77.878, -91.073, -127.344, -49.123, 94.526, 12.157]
  Set speed (100.0 mm/s)
  Smooth(1)
  MoveL 97 to (1.98, 50.31, -0.65) mm, rotated rx 0 ry 85.03 rz -0.76 deg; joints [-78.149, -91.465, -126.734, -50.034, 94.712, 11.89]
  MoveL 98 to (2.06, 49.53, -1.69) mm, rotated rx 0 ry 85.35 rz 0.15 deg; joints [-78.235, -91.924, -125.952, -51.324, 94.584, 11.803]
  MoveL 99 to (2.12, 48.9, -2.48) mm, rotated rx 0 ry 85.74 rz 1.06 deg; joints [-78.244, -92.363, -125.193, -52.612, 94.385, 11.789]
  MoveL 100 to (2.19, 48.24, -3.26) mm, rotated rx 0 ry 86.29 rz 2.06 deg; joints [-78.175, -92.845, -124.358, -54.054, 94.055, 11.848]
  MoveL 101 to (2.26, 47.54, -4.04) mm, rotated rx 0 ry 87 rz 3.15 deg; joints [-78.025, -93.372, -123.453, -55.632, 93.584, 11.981]
  MoveL 102 to (2.33, 46.83, -4.81) mm, rotated rx 0 ry 87.85 rz 4.27 deg; joints [-77.809, -93.929, -122.513, -57.28, 93.002, 12.173]
  MoveL 103 to (2.41, 46.1, -5.55) mm, rotated rx 0 ry 88.8 rz 5.43 deg; joints [-77.549, -94.521, -121.541, -58.982, 92.345, 12.405]
  MoveL 104 to (2.5, 45.3, -6.35) mm, rotated rx 0 ry 89.92 rz 6.69 deg; joints [-77.22, -95.187, -120.48, -60.84, 91.555, 12.696]
  MoveL 105 to (2.6, 44.41, -7.18) mm, rotated rx 180 ry 88.78 rz -171.99 deg; joints [-76.821, -95.918, -119.355, -62.808, 90.629, 13.049]
  MoveL 106 to (2.71, 43.5, -8) mm, rotated rx 180 ry 87.4 rz -170.72 deg; joints [-76.385, -96.651, -118.269, -64.708, 89.644, 13.433]
  MoveL 107 to (2.81, 42.61, -8.78) mm, rotated rx -180 ry 86.02 rz -169.55 deg; joints [-75.946, -97.362, -117.254, -66.482, 88.66, 13.82]
  MoveL 108 to (2.92, 41.72, -9.51) mm, rotated rx 180 ry 84.67 rz -168.46 deg; joints [-75.514, -98.047, -116.311, -68.129, 87.697, 14.199]
  MoveL 109 to (3.02, 40.83, -10.23) mm, rotated rx 180 ry 83.3 rz -167.43 deg; joints [-75.077, -98.727, -115.407, -69.707, 86.728, 14.582]
  MoveL 110 to (3.14, 39.86, -10.98) mm, rotated rx -180 ry 81.82 rz -166.42 deg; joints [-74.596, -99.426, -114.51, -71.286, 85.67, 15.008]
  MoveL 111 to (3.26, 38.88, -11.71) mm, rotated rx -180 ry 80.31 rz -165.48 deg; joints [-74.104, -100.112, -113.664, -72.788, 84.595, 15.446]
  MoveL 112 to (3.38, 37.89, -12.42) mm, rotated rx -180 ry 78.77 rz -164.61 deg; joints [-73.596, -100.776, -112.879, -74.204, 83.493, 15.905]
  MoveL 113 to (3.5, 36.94, -13.07) mm, rotated rx 180 ry 77.32 rz -163.85 deg; joints [-73.12, -101.388, -112.18, -75.476, 82.46, 16.339]
  MoveL 114 to (3.62, 35.99, -13.7) mm, rotated rx -180 ry 75.89 rz -163.15 deg; joints [-72.65, -101.976, -111.537, -76.662, 81.435, 16.776]
  MoveL 115 to (3.74, 35.01, -14.32) mm, rotated rx 180 ry 74.48 rz -162.54 deg; joints [-72.19, -102.527, -110.96, -77.745, 80.429, 17.211]
  MoveL 116 to (3.87, 34.03, -14.91) mm, rotated rx -180 ry 73.13 rz -162.02 deg; joints [-71.746, -103.033, -110.455, -78.706, 79.452, 17.641]
  MoveL 117 to (3.99, 33.04, -15.49) mm, rotated rx 180 ry 71.85 rz -161.62 deg; joints [-71.327, -103.485, -110.03, -79.532, 78.516, 18.062]
  MoveL 118 to (4.12, 32.05, -16.04) mm, rotated rx -180 ry 70.68 rz -161.31 deg; joints [-70.944, -103.876, -109.686, -80.211, 77.647, 18.459]
  MoveL 119 to (4.25, 31.06, -16.56) mm, rotated rx -180 ry 69.59 rz -161.15 deg; joints [-70.577, -104.194, -109.438, -80.726, 76.808, 18.859]
  MoveL 120 to (4.37, 30.12, -17.03) mm, rotated rx -180 ry 68.65 rz -161.1 deg; joints [-70.257, -104.431, -109.283, -81.072, 76.066, 19.225]
  MoveL 121 to (4.5, 29.18, -17.48) mm, rotated rx 180 ry 67.76 rz -161.19 deg; joints [-69.942, -104.596, -109.223, -81.262, 75.332, 19.61]
  MoveL 122 to (4.62, 28.23, -17.9) mm, rotated rx -180 ry 66.91 rz -161.44 deg; joints [-69.625, -104.684, -109.265, -81.288, 74.597, 20.02]
  MoveL 123 to (4.74, 27.31, -18.29) mm, rotated rx -180 ry 66.25 rz -161.57 deg; joints [-69.396, -104.808, -109.235, -81.372, 74.025, 20.321]
  MoveL 124 to (4.91, 25.97, -18.81) mm, rotated rx 180 ry 65.26 rz -162.24 deg; joints [-68.988, -104.754, -109.516, -81.018, 73.066, 20.913]
  MoveL 125 to (5.08, 24.62, -19.29) mm, rotated rx 180 ry 64.41 rz -163.14 deg; joints [-68.596, -104.586, -109.945, -80.402, 72.138, 21.527]
  MoveL 126 to (5.25, 23.24, -19.71) mm, rotated rx -180 ry 63.76 rz -163.93 deg; joints [-68.303, -104.453, -110.299, -79.822, 71.393, 22.014]
  MoveL 127 to (5.43, 21.89, -20.07) mm, rotated rx 180 ry 63.29 rz -164.53 deg; joints [-68.11, -104.397, -110.52, -79.379, 70.837, 22.359]
  MoveL 128 to (5.61, 20.58, -20.37) mm, rotated rx 180 ry 62.94 rz -164.92 deg; joints [-67.99, -104.429, -110.598, -79.112, 70.432, 22.584]
  MoveL 129 to (5.8, 19.35, -20.59) mm, rotated rx 180 ry 62.66 rz -165.06 deg; joints [-67.927, -104.562, -110.523, -79.066, 70.15, 22.707]
  MoveL 130 to (6.01, 18.15, -20.76) mm, rotated rx 180 ry 62.38 rz -165 deg; joints [-67.889, -104.787, -110.317, -79.221, 69.93, 22.773]
  MoveL 131 to (6.25, 17, -20.88) mm, rotated rx -180 ry 62.07 rz -164.79 deg; joints [-67.852, -105.09, -110.011, -79.549, 69.725, 22.82]
  MoveL 132 to (6.49, 15.91, -20.95) mm, rotated rx -180 ry 61.69 rz -164.4 deg; joints [-67.808, -105.484, -109.591, -80.088, 69.528, 22.851]
  MoveL 133 to (6.77, 14.83, -20.97) mm, rotated rx -180 ry 61.19 rz -163.89 deg; joints [-67.733, -105.957, -109.087, -80.795, 69.283, 22.905]
  MoveL 134 to (7.09, 13.76, -20.94) mm, rotated rx 180 ry 60.57 rz -163.28 deg; joints [-67.614, -106.495, -108.527, -81.638, 68.967, 23.004]
  MoveL 135 to (7.44, 12.71, -20.87) mm, rotated rx 180 ry 59.81 rz -162.64 deg; joints [-67.442, -107.074, -107.948, -82.57, 68.566, 23.163]
  MoveL 136 to (7.81, 11.72, -20.75) mm, rotated rx 180 ry 59 rz -162.47 deg; joints [-67.175, -107.433, -107.699, -83.043, 68, 23.512]
  MoveL 137 to (7.95, 11.39, -20.7) mm, rotated rx 180 ry 58.75 rz -162.76 deg; joints [-67.044, -107.386, -107.849, -82.847, 67.734, 23.736]
  Set speed (1000.0 mm/s)
  MoveL 138 to (7.95, 11.39, -20.7) mm, rotated rx -180 ry 58.75 rz -162.76 deg; joints [-67.044, -107.386, -107.849, -82.847, 67.734, 23.736]
  MoveL 139 to (-73.7, -13.94, 31.18) mm, rotated rx 180 ry 58.75 rz -162.76 deg; joints [-63.241, -106.587, -95.037, -97.762, 69.563, 27.316]
  Set speed (1000.0 mm/s)
  MoveL 140 to (-97.68, 19.69, -50.49) mm, rotated rx 0 ry 86.28 rz 3.56 deg; joints [-84.828, -90.754, -109.371, -73.085, 94.029, 5.175]
  MoveL 141 to (1.91, 25.89, -44) mm, rotated rx 0 ry 86.28 rz 3.56 deg; joints [-83.955, -96.783, -119.419, -56.946, 94.077, 6.049]
  MoveL 142 to (1.91, 25.89, -44) mm, rotated rx 0 ry 86.28 rz 3.56 deg; joints [-83.955, -96.783, -119.419, -56.946, 94.077, 6.049]
  Set speed (100.0 mm/s)
  Smooth(1)
  MoveL 143 to (1.98, 24.59, -43.9) mm, rotated rx 0 ry 86.86 rz 3.93 deg; joints [-83.674, -97.056, -118.985, -57.523, 93.555, 6.323]
  MoveL 144 to (2.06, 23.31, -43.74) mm, rotated rx 0 ry 87.81 rz 4.11 deg; joints [-83.186, -97.213, -118.716, -57.889, 92.662, 6.804]
  MoveL 145 to (2.12, 22.3, -43.59) mm, rotated rx 0 ry 88.79 rz 4.22 deg; joints [-82.678, -97.313, -118.531, -58.185, 91.74, 7.305]
  MoveL 146 to (2.19, 21.29, -43.41) mm, rotated rx 0 ry 89.93 rz 4.24 deg; joints [-82.08, -97.373, -118.416, -58.405, 90.656, 7.898]
  MoveL 147 to (2.26, 20.27, -43.2) mm, rotated rx -180 ry 88.78 rz -175.83 deg; joints [-81.394, -97.394, -118.378, -58.533, 89.414, 8.584]
  MoveL 148 to (2.33, 19.25, -42.96) mm, rotated rx -180 ry 87.38 rz -176 deg; joints [-80.646, -97.384, -118.411, -58.578, 88.064, 9.336]
  MoveL 149 to (2.41, 18.24, -42.7) mm, rotated rx -180 ry 85.9 rz -176.23 deg; joints [-79.851, -97.359, -118.491, -58.577, 86.631, 10.144]
  MoveL 150 to (2.5, 17.15, -42.4) mm, rotated rx -180 ry 84.25 rz -176.57 deg; joints [-78.954, -97.317, -118.639, -58.509, 85.013, 11.069]
  MoveL 151 to (2.6, 15.98, -42.05) mm, rotated rx -180 ry 82.45 rz -177.04 deg; joints [-77.966, -97.256, -118.866, -58.352, 83.234, 12.103]
  MoveL 152 to (2.71, 14.82, -41.67) mm, rotated rx -180 ry 80.66 rz -177.61 deg; joints [-76.975, -97.184, -119.159, -58.106, 81.445, 13.163]
  MoveL 153 to (2.81, 13.7, -41.29) mm, rotated rx 180 ry 78.96 rz -178.23 deg; joints [-76.019, -97.115, -119.485, -57.814, 79.721, 14.207]
  MoveL 154 to (2.92, 12.62, -40.89) mm, rotated rx -180 ry 77.35 rz -178.88 deg; joints [-75.108, -97.056, -119.828, -57.493, 78.073, 15.225]
  MoveL 155 to (3.02, 11.55, -40.47) mm, rotated rx -180 ry 75.79 rz -179.59 deg; joints [-74.212, -97.004, -120.198, -57.137, 76.45, 16.252]
  MoveL 156 to (3.14, 10.42, -40.01) mm, rotated rx -180 ry 74.19 rz 179.58 deg; joints [-73.28, -96.942, -120.641, -56.671, 74.757, 17.348]
  MoveL 157 to (3.26, 9.3, -39.53) mm, rotated rx 180 ry 72.65 rz 178.67 deg; joints [-72.364, -96.883, -121.123, -56.142, 73.086, 18.456]
  MoveL 158 to (3.38, 8.19, -39.02) mm, rotated rx -180 ry 71.17 rz 177.67 deg; joints [-71.465, -96.82, -121.654, -55.523, 71.44, 19.576]
  MoveL 159 to (3.5, 7.16, -38.53) mm, rotated rx -180 ry 69.83 rz 176.68 deg; joints [-70.637, -96.772, -122.172, -54.904, 69.919, 20.635]
  MoveL 160 to (3.62, 6.13, -38.01) mm, rotated rx -180 ry 68.57 rz 175.65 deg; joints [-69.841, -96.73, -122.707, -54.237, 68.448, 21.683]
  MoveL 161 to (3.74, 5.11, -37.48) mm, rotated rx -180 ry 67.41 rz 174.59 deg; joints [-69.086, -96.697, -123.253, -53.522, 67.049, 22.702]
  MoveL 162 to (3.87, 4.1, -36.93) mm, rotated rx -180 ry 66.37 rz 173.51 deg; joints [-68.383, -96.669, -123.801, -52.758, 65.742, 23.671]
  MoveL 163 to (3.99, 3.1, -36.36) mm, rotated rx 180 ry 65.46 rz 172.43 deg; joints [-67.742, -96.647, -124.341, -51.954, 64.549, 24.572]
  MoveL 164 to (4.12, 2.14, -35.78) mm, rotated rx 180 ry 64.71 rz 171.39 deg; joints [-67.177, -96.633, -124.853, -51.141, 63.497, 25.376]
  MoveL 165 to (4.25, 1.18, -35.18) mm, rotated rx -180 ry 64.11 rz 170.36 deg; joints [-66.681, -96.611, -125.369, -50.248, 62.575, 26.083]
  MoveL 166 to (4.37, 0.31, -34.6) mm, rotated rx 180 ry 63.69 rz 169.43 deg; joints [-66.28, -96.587, -125.838, -49.376, 61.836, 26.65]
  MoveL 167 to (4.5, -0.55, -34.01) mm, rotated rx 180 ry 63.41 rz 168.48 deg; joints [-65.938, -96.545, -126.325, -48.4, 61.211, 27.12]
  MoveL 168 to (4.62, -1.39, -33.4) mm, rotated rx -180 ry 63.28 rz 167.51 deg; joints [-65.654, -96.481, -126.84, -47.297, 60.705, 27.485]
  MoveL 169 to (4.74, -2.19, -32.8) mm, rotated rx 180 ry 63.13 rz 166.77 deg; joints [-65.405, -96.476, -127.203, -46.485, 60.266, 27.813]
  MoveL 170 to (4.91, -3.31, -31.9) mm, rotated rx -180 ry 63.31 rz 165.49 deg; joints [-65.171, -96.357, -127.919, -44.76, 59.893, 28.029]
  MoveL 171 to (5.08, -4.4, -30.96) mm, rotated rx -180 ry 63.73 rz 164.26 deg; joints [-65.043, -96.22, -128.637, -42.898, 59.741, 28.046]
  MoveL 172 to (5.25, -5.45, -29.99) mm, rotated rx -180 ry 64.15 rz 163.29 deg; joints [-64.96, -96.145, -129.18, -41.361, 59.693, 28.005]
  MoveL 173 to (5.43, -6.44, -28.99) mm, rotated rx 180 ry 64.46 rz 162.58 deg; joints [-64.884, -96.137, -129.54, -40.227, 59.67, 27.982]
  MoveL 174 to (5.61, -7.35, -28) mm, rotated rx -180 ry 64.65 rz 162.08 deg; joints [-64.788, -96.183, -129.755, -39.458, 59.613, 28.024]
  MoveL 175 to (5.8, -8.16, -27.05) mm, rotated rx -180 ry 64.66 rz 161.74 deg; joints [-64.647, -96.275, -129.851, -39.032, 59.466, 28.17]
  MoveL 176 to (6.01, -8.91, -26.1) mm, rotated rx -180 ry 64.51 rz 161.47 deg; joints [-64.448, -96.404, -129.881, -38.83, 59.206, 28.431]
  MoveL 177 to (6.25, -9.59, -25.16) mm, rotated rx 180 ry 64.22 rz 161.22 deg; joints [-64.186, -96.559, -129.89, -38.756, 58.821, 28.808]
  MoveL 178 to (6.49, -10.19, -24.25) mm, rotated rx -180 ry 63.76 rz 160.97 deg; joints [-63.849, -96.743, -129.883, -38.816, 58.281, 29.329]
  MoveL 179 to (6.77, -10.75, -23.33) mm, rotated rx -180 ry 63.16 rz 160.65 deg; joints [-63.433, -96.951, -129.906, -38.897, 57.581, 29.992]
  MoveL 180 to (7.09, -11.26, -22.39) mm, rotated rx 180 ry 62.44 rz 160.2 deg; joints [-62.941, -97.179, -129.985, -38.932, 56.728, 30.793]
  MoveL 181 to (7.44, -11.72, -21.44) mm, rotated rx -180 ry 61.65 rz 159.62 deg; joints [-62.39, -97.417, -130.143, -38.865, 55.749, 31.707]
  MoveL 182 to (7.81, -12.11, -20.53) mm, rotated rx -180 ry 61.24 rz 158.8 deg; joints [-61.946, -97.558, -130.52, -38.18, 54.992, 32.367]
  MoveL 183 to (7.95, -12.23, -20.22) mm, rotated rx -180 ry 61.39 rz 158.44 deg; joints [-61.895, -97.535, -130.762, -37.568, 54.946, 32.357]
  Set speed (1000.0 mm/s)
  MoveL 184 to (7.95, -12.23, -20.22) mm, rotated rx -180 ry 61.39 rz 158.44 deg; joints [-61.895, -97.535, -130.762, -37.568, 54.946, 32.357]
  MoveL 185 to (-73.7, 20.03, 27.66) mm, rotated rx 180 ry 61.39 rz 158.44 deg; joints [-53.652, -85.124, -126.194, -60.362, 54.769, 42.44]
  Set speed (1000.0 mm/s)
  MoveL 186 to (-97.68, -33.88, -42.3) mm, rotated rx 180 ry 88.79 rz -175 deg; joints [-82.245, -98.245, -100.722, -76.155, 89.471, 7.726]
  MoveL 187 to (1.91, -25.16, -44.42) mm, rotated rx 180 ry 88.79 rz -175 deg; joints [-82.347, -103.384, -110.714, -61.024, 89.462, 7.624]
  MoveL 188 to (1.91, -25.16, -44.42) mm, rotated rx 180 ry 88.79 rz -175 deg; joints [-82.347, -103.384, -110.714, -61.024, 89.462, 7.624]
  Set speed (100.0 mm/s)
  Smooth(1)
  MoveL 189 to (1.98, -25.72, -43.25) mm, rotated rx -180 ry 88.17 rz -175.31 deg; joints [-81.917, -103.281, -110.916, -60.701, 88.848, 8.058]
  MoveL 190 to (2.06, -26.23, -42.05) mm, rotated rx -180 ry 87.54 rz -176.05 deg; joints [-81.447, -102.999, -111.451, -59.824, 88.159, 8.537]
  MoveL 191 to (2.12, -26.6, -41.1) mm, rotated rx 180 ry 86.96 rz -176.84 deg; joints [-81.012, -102.688, -112.044, -58.867, 87.487, 8.983]
  MoveL 192 to (2.19, -26.95, -40.14) mm, rotated rx -180 ry 86.36 rz -177.81 deg; joints [-80.553, -102.307, -112.782, -57.666, 86.769, 9.455]
  MoveL 193 to (2.26, -27.27, -39.15) mm, rotated rx 180 ry 85.78 rz -178.97 deg; joints [-80.073, -101.863, -113.665, -56.211, 86.018, 9.949]
  MoveL 194 to (2.33, -27.58, -38.15) mm, rotated rx -180 ry 85.23 rz 179.73 deg; joints [-79.588, -101.382, -114.652, -54.562, 85.257, 10.448]
  MoveL 195 to (2.41, -27.86, -37.15) mm, rotated rx -180 ry 84.7 rz 178.32 deg; joints [-79.091, -100.882, -115.716, -52.764, 84.475, 10.956]
  MoveL 196 to (2.5, -28.14, -36.05) mm, rotated rx 180 ry 84.17 rz 176.71 deg; joints [-78.555, -100.335, -116.934, -50.67, 83.634, 11.498]
  MoveL 197 to (2.6, -28.42, -34.87) mm, rotated rx 180 ry 83.68 rz 174.91 deg; joints [-77.994, -99.76, -118.291, -48.286, 82.764, 12.055]
  MoveL 198 to (2.71, -28.68, -33.67) mm, rotated rx 180 ry 83.29 rz 173.07 deg; joints [-77.461, -99.215, -119.669, -45.804, 81.95, 12.572]
  MoveL 199 to (2.81, -28.9, -32.51) mm, rotated rx 180 ry 82.99 rz 171.27 deg; joints [-76.965, -98.727, -121.004, -43.341, 81.207, 13.037]
  MoveL 200 to (2.92, -29.1, -31.38) mm, rotated rx -180 ry 82.76 rz 169.54 deg; joints [-76.507, -98.302, -122.279, -40.926, 80.532, 13.452]
  MoveL 201 to (3.02, -29.28, -30.24) mm, rotated rx -180 ry 82.6 rz 167.83 deg; joints [-76.069, -97.924, -123.535, -38.486, 79.901, 13.83]
  MoveL 202 to (3.14, -29.44, -29.03) mm, rotated rx 180 ry 82.53 rz 166.03 deg; joints [-75.647, -97.576, -124.848, -35.849, 79.318, 14.17]
  MoveL 203 to (3.26, -29.58, -27.82) mm, rotated rx 180 ry 82.54 rz 164.24 deg; joints [-75.259, -97.285, -126.139, -33.169, 78.805, 14.456]
  MoveL 204 to (3.38, -29.7, -26.61) mm, rotated rx 180 ry 82.64 rz 162.47 deg; joints [-74.915, -97.054, -127.408, -30.437, 78.382, 14.676]
  MoveL 205 to (3.5, -29.79, -25.46) mm, rotated rx -180 ry 82.8 rz 160.83 deg; joints [-74.617, -96.894, -128.571, -27.849, 78.038, 14.84]
  MoveL 206 to (3.62, -29.86, -24.31) mm, rotated rx -180 ry 83.02 rz 159.24 deg; joints [-74.355, -96.793, -129.685, -25.279, 77.768, 14.953]
  MoveL 207 to (3.74, -29.91, -23.17) mm, rotated rx 180 ry 83.3 rz 157.74 deg; joints [-74.134, -96.749, -130.735, -22.765, 77.582, 15.015]
  MoveL 208 to (3.87, -29.93, -22.02) mm, rotated rx -180 ry 83.65 rz 156.33 deg; joints [-73.958, -96.757, -131.707, -20.348, 77.489, 15.026]
  MoveL 209 to (3.99, -29.93, -20.87) mm, rotated rx 180 ry 84.04 rz 155.05 deg; joints [-73.829, -96.811, -132.586, -18.074, 77.492, 14.99]
  MoveL 210 to (4.12, -29.91, -19.74) mm, rotated rx -180 ry 84.47 rz 153.92 deg; joints [-73.743, -96.896, -133.355, -16.011, 77.578, 14.92]
  MoveL 211 to (4.25, -29.87, -18.61) mm, rotated rx -180 ry 84.96 rz 152.92 deg; joints [-73.719, -97.006, -134.029, -14.123, 77.793, 14.797]
  MoveL 212 to (4.37, -29.81, -17.57) mm, rotated rx -180 ry 85.46 rz 152.12 deg; joints [-73.743, -97.12, -134.568, -12.545, 78.083, 14.65]
  MoveL 213 to (4.5, -29.73, -16.53) mm, rotated rx 180 ry 86.04 rz 151.44 deg; joints [-73.833, -97.242, -135.03, -11.122, 78.509, 14.451]
  MoveL 214 to (4.62, -29.62, -15.5) mm, rotated rx 180 ry 86.7 rz 150.87 deg; joints [-73.998, -97.367, -135.414, -9.857, 79.087, 14.196]
  MoveL 215 to (4.74, -29.5, -14.5) mm, rotated rx -180 ry 87.18 rz 150.39 deg; joints [-74.072, -97.477, -135.742, -8.814, 79.471, 14.045]
  MoveL 216 to (4.91, -29.28, -13.09) mm, rotated rx 180 ry 88.24 rz 149.93 deg; joints [-74.448, -97.635, -136.063, -7.564, 80.568, 13.603]
  MoveL 217 to (5.08, -29.01, -11.67) mm, rotated rx -180 ry 89.39 rz 149.67 deg; joints [-74.922, -97.775, -136.25, -6.652, 81.862, 13.11]
  MoveL 218 to (5.25, -28.69, -10.28) mm, rotated rx 0 ry 89.65 rz -30.47 deg; joints [-75.291, -97.882, -136.371, -6.028, 82.943, 12.739]
  MoveL 219 to (5.43, -28.33, -8.92) mm, rotated rx 0 ry 88.94 rz -30.56 deg; joints [-75.515, -97.958, -136.475, -5.578, 83.724, 12.514]
  MoveL 220 to (5.61, -27.93, -7.64) mm, rotated rx 0 ry 88.47 rz -30.67 deg; joints [-75.601, -98.011, -136.597, -5.189, 84.212, 12.415]
  MoveL 221 to (5.8, -27.51, -6.46) mm, rotated rx 0 ry 88.21 rz -30.83 deg; joints [-75.55, -98.053, -136.768, -4.762, 84.404, 12.433]
  MoveL 222 to (6.01, -27.06, -5.34) mm, rotated rx 0 ry 88.1 rz -31.09 deg; joints [-75.397, -98.099, -137.005, -4.216, 84.378, 12.53]
  MoveL 223 to (6.25, -26.58, -4.28) mm, rotated rx 0 ry 88.08 rz -31.46 deg; joints [-75.175, -98.164, -137.315, -3.496, 84.202, 12.673]
  MoveL 224 to (6.49, -26.1, -3.3) mm, rotated rx 0 ry 88.16 rz -31.96 deg; joints [-74.879, -98.26, -137.715, -2.547, 83.858, 12.861]
  MoveL 225 to (6.77, -25.58, -2.36) mm, rotated rx 0 ry 88.26 rz -32.63 deg; joints [-74.54, -98.407, -138.21, -1.313, 83.428, 13.061]
  MoveL 226 to (7.09, -25.02, -1.44) mm, rotated rx 0 ry 88.36 rz -33.44 deg; joints [-74.186, -98.622, -138.795, 0.228, 82.964, 13.246]
  MoveL 227 to (7.44, -24.43, -0.58) mm, rotated rx 0 ry 88.39 rz -34.38 deg; joints [-73.849, -98.918, -139.451, 2.06, 82.525, 13.388]
  MoveL 228 to (7.81, -23.83, 0.22) mm, rotated rx 0 ry 88.06 rz -35.14 deg; joints [-73.803, -99.233, -139.977, 3.713, 82.655, 13.297]
  MoveL 229 to (7.95, -23.62, 0.48) mm, rotated rx 0 ry 87.71 rz -35.2 deg; joints [-73.979, -99.307, -140.036, 4.009, 83.077, 13.131]
  Set speed (1000.0 mm/s)
  MoveL 230 to (7.95, -23.62, 0.48) mm, rotated rx 0 ry 87.71 rz -35.2 deg; joints [-73.979, -99.307, -140.036, 4.009, 83.077, 13.131]
  MoveL 231 to (-73.7, 33.97, -3.52) mm, rotated rx 0 ry 87.71 rz -35.2 deg; joints [-71.575, -77.196, -142.491, -15.911, 81.715, 15.129]
  Set speed (1000.0 mm/s)
  MoveL 232 to (-97.61, -52.9, 9.17) mm, rotated rx -180 ry 84.5 rz -178.94 deg; joints [-74.841, -98.665, -100.94, -72.865, 84.966, 15.216]
  MoveL 233 to (1.91, -51.05, -0.42) mm, rotated rx -180 ry 84.5 rz -178.94 deg; joints [-75.801, -104.706, -109.792, -57.887, 84.926, 14.254]
  MoveL 234 to (1.91, -51.05, -0.42) mm, rotated rx -180 ry 84.5 rz -178.94 deg; joints [-75.801, -104.706, -109.792, -57.887, 84.926, 14.254]
  Set speed (100.0 mm/s)
  Smooth(1)
  MoveL 235 to (1.98, -50.31, 0.65) mm, rotated rx -180 ry 84.49 rz -179.64 deg; joints [-75.584, -104.348, -110.467, -56.909, 84.755, 14.477]
  MoveL 236 to (2.06, -49.53, 1.69) mm, rotated rx 180 ry 84.93 rz 179.51 deg; joints [-75.554, -103.928, -111.275, -55.593, 84.972, 14.503]
  MoveL 237 to (2.12, -48.9, 2.48) mm, rotated rx 180 ry 85.33 rz 178.59 deg; joints [-75.52, -103.505, -112.12, -54.18, 85.121, 14.529]
  MoveL 238 to (2.19, -48.24, 3.26) mm, rotated rx 180 ry 85.86 rz 177.56 deg; joints [-75.544, -103.051, -113.054, -52.565, 85.386, 14.491]
  MoveL 239 to (2.26, -47.54, 4.04) mm, rotated rx -180 ry 86.58 rz 176.45 deg; joints [-75.641, -102.583, -114.054, -50.777, 85.807, 14.37]
  MoveL 240 to (2.33, -46.83, 4.81) mm, rotated rx -180 ry 87.43 rz 175.32 deg; joints [-75.804, -102.124, -115.084, -48.881, 86.363, 14.177]
  MoveL 241 to (2.41, -46.1, 5.55) mm, rotated rx 180 ry 88.35 rz 174.12 deg; joints [-75.998, -101.669, -116.162, -46.856, 86.981, 13.947]
  MoveL 242 to (2.5, -45.3, 6.35) mm, rotated rx -180 ry 89.44 rz 172.8 deg; joints [-76.259, -101.207, -117.338, -44.591, 87.751, 13.642]
  MoveL 243 to (2.6, -44.41, 7.18) mm, rotated rx 0 ry 89.29 rz -8.58 deg; joints [-76.603, -100.766, -118.571, -42.145, 88.71, 13.248]
  MoveL 244 to (2.71, -43.5, 8) mm, rotated rx 0 ry 87.92 rz -9.88 deg; joints [-77.023, -100.402, -119.728, -39.773, 89.822, 12.781]
  MoveL 245 to (2.81, -42.61, 8.78) mm, rotated rx 0 ry 86.55 rz -11.09 deg; joints [-77.471, -100.113, -120.798, -37.522, 90.981, 12.293]
  MoveL 246 to (2.92, -41.72, 9.51) mm, rotated rx 0 ry 85.23 rz -12.24 deg; joints [-77.917, -99.885, -121.803, -35.362, 92.126, 11.813]
  MoveL 247 to (3.02, -40.83, 10.23) mm, rotated rx 0 ry 83.93 rz -13.38 deg; joints [-78.368, -99.703, -122.786, -33.206, 93.278, 11.331]
  MoveL 248 to (3.14, -39.86, 10.98) mm, rotated rx 0 ry 82.48 rz -14.46 deg; joints [-78.915, -99.595, -123.715, -31.085, 94.641, 10.765]
  MoveL 249 to (3.26, -38.88, 11.71) mm, rotated rx 0 ry 81 rz -15.48 deg; joints [-79.494, -99.552, -124.583, -29.043, 96.068, 10.178]
  MoveL 250 to (3.38, -37.89, 12.42) mm, rotated rx 0 ry 79.46 rz -16.39 deg; joints [-80.135, -99.587, -125.341, -27.174, 97.623, 9.546]
  MoveL 251 to (3.5, -36.94, 13.07) mm, rotated rx 0 ry 78.04 rz -17.23 deg; joints [-80.735, -99.663, -126.033, -25.433, 99.081, 8.959]
  MoveL 252 to (3.62, -35.99, 13.7) mm, rotated rx 0 ry 76.63 rz -18.01 deg; joints [-81.346, -99.787, -126.658, -23.807, 100.561, 8.37]
  MoveL 253 to (3.74, -35.01, 14.32) mm, rotated rx 0 ry 75.26 rz -18.71 deg; joints [-81.956, -99.95, -127.211, -22.324, 102.04, 7.789]
  MoveL 254 to (3.87, -34.03, 14.91) mm, rotated rx 0 ry 73.92 rz -19.3 deg; joints [-82.557, -100.145, -127.681, -21.022, 103.501, 7.223]
  MoveL 255 to (3.99, -33.04, 15.49) mm, rotated rx 0 ry 72.64 rz -19.77 deg; joints [-83.142, -100.36, -128.056, -19.95, 104.928, 6.679]
  MoveL 256 to (4.12, -32.05, 16.04) mm, rotated rx 0 ry 71.5 rz -20.19 deg; joints [-83.662, -100.568, -128.391, -19.004, 106.213, 6.195]
  MoveL 257 to (4.25, -31.06, 16.56) mm, rotated rx 0 ry 70.39 rz -20.4 deg; joints [-84.177, -100.783, -128.593, -18.399, 107.489, 5.722]
  MoveL 258 to (4.37, -30.12, 17.03) mm, rotated rx 0 ry 69.51 rz -20.65 deg; joints [-84.574, -100.955, -128.815, -17.796, 108.495, 5.354]
  MoveL 259 to (4.5, -29.18, 17.48) mm, rotated rx 0 ry 68.67 rz -20.75 deg; joints [-84.96, -101.122, -128.948, -17.439, 109.475, 4.999]
  MoveL 260 to (4.62, -28.23, 17.9) mm, rotated rx 0 ry 67.82 rz -20.61 deg; joints [-85.36, -101.288, -128.932, -17.481, 110.483, 4.636]
  MoveL 261 to (4.74, -27.31, 18.29) mm, rotated rx 0 ry 67.59 rz -21.65 deg; joints [-85.382, -101.325, -129.69, -15.654, 110.647, 4.587]
  MoveL 262 to (4.91, -25.97, 18.81) mm, rotated rx 0 ry 66.62 rz -21.34 deg; joints [-85.836, -101.495, -129.614, -15.942, 111.811, 4.177]
  MoveL 263 to (5.08, -24.62, 19.29) mm, rotated rx 0 ry 65.56 rz -20.32 deg; joints [-86.364, -101.663, -129.096, -17.429, 113.132, 3.708]
  MoveL 264 to (5.25, -23.24, 19.71) mm, rotated rx 0 ry 64.66 rz -19.21 deg; joints [-86.803, -101.793, -128.548, -19.064, 114.247, 3.311]
  MoveL 265 to (5.43, -21.89, 20.07) mm, rotated rx 0 ry 63.96 rz -18.23 deg; joints [-87.137, -101.882, -128.101, -20.489, 115.112, 3.003]
  MoveL 266 to (5.61, -20.58, 20.37) mm, rotated rx 0 ry 63.41 rz -17.46 deg; joints [-87.391, -101.941, -127.785, -21.595, 115.781, 2.764]
  MoveL 267 to (5.8, -19.35, 20.59) mm, rotated rx 0 ry 62.98 rz -17.03 deg; joints [-87.581, -101.975, -127.681, -22.155, 116.285, 2.58]
  MoveL 268 to (6.01, -18.15, 20.76) mm, rotated rx 0 ry 62.59 rz -16.83 deg; joints [-87.755, -102.006, -127.712, -22.355, 116.741, 2.406]
  MoveL 269 to (6.25, -17, 20.88) mm, rotated rx 0 ry 62.17 rz -16.76 deg; joints [-87.945, -102.052, -127.812, -22.351, 117.216, 2.213]
  MoveL 270 to (6.49, -15.91, 20.95) mm, rotated rx 0 ry 61.72 rz -17.01 deg; joints [-88.154, -102.124, -128.087, -21.84, 117.721, 1.994]
  MoveL 271 to (6.77, -14.83, 20.97) mm, rotated rx 0 ry 61.17 rz -17.4 deg; joints [-88.419, -102.246, -128.428, -21.106, 118.343, 1.714]
  MoveL 272 to (7.09, -13.76, 20.94) mm, rotated rx 0 ry 60.5 rz -17.87 deg; joints [-88.753, -102.432, -128.793, -20.239, 119.11, 1.359]
  MoveL 273 to (7.44, -12.71, 20.87) mm, rotated rx 0 ry 59.7 rz -18.39 deg; joints [-89.155, -102.689, -129.157, -19.299, 120.027, 0.926]
  MoveL 274 to (7.81, -11.72, 20.75) mm, rotated rx 0 ry 58.95 rz -17.87 deg; joints [-89.546, -102.898, -128.916, -20.059, 120.91, 0.504]
  MoveL 275 to (7.95, -11.39, 20.7) mm, rotated rx 0 ry 58.8 rz -16.9 deg; joints [-89.631, -102.904, -128.393, -21.594, 121.095, 0.413]
  Set speed (1000.0 mm/s)
  MoveL 276 to (7.95, -11.39, 20.7) mm, rotated rx 0 ry 58.8 rz -16.9 deg; joints [-89.631, -102.904, -128.393, -21.594, 121.095, 0.413]
  MoveL 277 to (-73.89, 13.47, -31.11) mm, rotated rx 0 ry 58.8 rz -16.9 deg; joints [-96.786, -91.463, -124.088, -41.669, 122.944, -7.742]

--- program hub (robot UR5) ---
  Smooth(1)
  Change Frame at (0, -480, 32.2) mm, rotated rx 0 ry 90 rz 0 deg
  Set Tool: laser_fixture_tool
  Show laser_fixture_tool
  Set speed (1000.0 mm/s)
  MoveJ 1 to (-70.79, -56.7, 38.74) mm, rotated rx 180 ry 71.65 rz -152.9 deg; joints [-70.169, -116.202, -80.363, -104.724, 81.4, 17.785]
  MoveL 2 to (-70.79, -56.7, 38.74) mm, rotated rx 180 ry 71.65 rz -152.9 deg; joints [-70.169, -116.202, -80.363, -104.724, 81.4, 17.785]
  MoveL 3 to (13.7, -13.47, 7.25) mm, rotated rx -180 ry 71.65 rz -152.9 deg; joints [-71.611, -114.797, -96.036, -90.261, 80.653, 16.536]
  MoveL 4 to (13.7, -13.47, 7.25) mm, rotated rx -180 ry 71.65 rz -152.9 deg; joints [-71.611, -114.797, -96.036, -90.261, 80.653, 16.536]
  Set speed (100.0 mm/s)
  Smooth(1)
  MoveL 5 to (13.7, -13.94, 6.31) mm, rotated rx -180 ry 73.47 rz -151.81 deg; joints [-72.538, -115.314, -95.153, -91.014, 82.213, 15.482]
  MoveL 6 to (13.7, -14.34, 5.34) mm, rotated rx -180 ry 75.36 rz -150.85 deg; joints [-73.471, -115.773, -94.371, -91.65, 83.785, 14.473]
  MoveL 7 to (13.7, -14.67, 4.34) mm, rotated rx -180 ry 77.3 rz -150.01 deg; joints [-74.407, -116.175, -93.693, -92.168, 85.369, 13.508]
  MoveL 8 to (13.7, -14.93, 3.33) mm, rotated rx -180 ry 79.28 rz -149.31 deg; joints [-75.345, -116.516, -93.123, -92.566, 86.96, 12.584]
  MoveL 9 to (13.7, -15.13, 2.3) mm, rotated rx -180 ry 81.31 rz -148.73 deg; joints [-76.284, -116.796, -92.664, -92.845, 88.557, 11.697]
  MoveL 10 to (13.7, -15.25, 1.25) mm, rotated rx -180 ry 83.36 rz -148.28 deg; joints [-77.221, -117.014, -92.317, -93.002, 90.158, 10.846]
  MoveL 11 to (13.7, -15.3, 0.21) mm, rotated rx 180 ry 85.44 rz -147.96 deg; joints [-78.154, -117.169, -92.084, -93.038, 91.76, 10.026]
  MoveL 12 to (13.7, -15.28, -0.84) mm, rotated rx -180 ry 87.53 rz -147.75 deg; joints [-79.082, -117.26, -91.967, -92.95, 93.362, 9.233]
  MoveL 13 to (13.7, -15.18, -1.89) mm, rotated rx 180 ry 89.63 rz -147.67 deg; joints [-80.004, -117.288, -91.967, -92.737, 94.961, 8.466]
  MoveL 14 to (13.7, -15.02, -2.92) mm, rotated rx 0 ry 88.27 rz 32.29 deg; joints [-80.917, -117.252, -92.083, -92.398, 96.554, 7.72]
  MoveL 15 to (13.7, -14.78, -3.95) mm, rotated rx 0 ry 86.17 rz 32.13 deg; joints [-81.819, -117.153, -92.316, -91.931, 98.139, 6.992]
  MoveL 16 to (13.7, -14.48, -4.95) mm, rotated rx 0 ry 84.09 rz 31.85 deg; joints [-82.709, -116.991, -92.665, -91.335, 99.714, 6.279]
  MoveL 17 to (13.7, -14.1, -5.93) mm, rotated rx 0 ry 82.03 rz 31.44 deg; joints [-83.586, -116.769, -93.128, -90.608, 101.276, 5.578]
  MoveL 18 to (13.7, -13.66, -6.88) mm, rotated rx 0 ry 79.99 rz 30.91 deg; joints [-84.446, -116.487, -93.703, -89.749, 102.822, 4.885]
  MoveL 19 to (13.7, -13.16, -7.8) mm, rotated rx 0 ry 77.99 rz 30.25 deg; joints [-85.288, -116.147, -94.388, -88.755, 104.348, 4.2]
  MoveL 20 to (13.7, -12.59, -8.69) mm, rotated rx 0 ry 76.03 rz 29.46 deg; joints [-86.111, -115.752, -95.18, -87.624, 105.852, 3.52]
  MoveL 21 to (13.7, -11.97, -9.53) mm, rotated rx 0 ry 74.13 rz 28.55 deg; joints [-86.911, -115.303, -96.075, -86.355, 107.329, 2.842]
  MoveL 22 to (13.7, -11.29, -10.33) mm, rotated rx 0 ry 72.28 rz 27.5 deg; joints [-87.687, -114.804, -97.071, -84.944, 108.775, 2.167]
  MoveL 23 to (13.7, -10.55, -11.08) mm, rotated rx 0 ry 70.5 rz 26.32 deg; joints [-88.436, -114.258, -98.162, -83.39, 110.185, 1.493]
  MoveL 24 to (13.7, -9.77, -11.78) mm, rotated rx 0 ry 68.8 rz 25 deg; joints [-89.156, -113.668, -99.344, -81.691, 111.555, 0.822]
  MoveL 25 to (13.7, -8.94, -12.42) mm, rotated rx 0 ry 67.18 rz 23.55 deg; joints [-89.844, -113.039, -100.612, -79.843, 112.88, 0.155]
  MoveL 26 to (13.7, -8.07, -13) mm, rotated rx 0 ry 65.66 rz 21.97 deg; joints [-90.498, -112.374, -101.96, -77.844, 114.152, -0.506]
  MoveL 27 to (13.7, -7.15, -13.52) mm, rotated rx 0 ry 64.24 rz 20.26 deg; joints [-91.114, -111.679, -103.384, -75.693, 115.365, -1.157]
  MoveL 28 to (13.7, -6.21, -13.98) mm, rotated rx 0 ry 62.94 rz 18.41 deg; joints [-91.69, -110.957, -104.876, -73.388, 116.512, -1.792]
  MoveL 29 to (13.7, -5.24, -14.37) mm, rotated rx 0 ry 61.76 rz 16.45 deg; joints [-92.222, -110.215, -106.431, -70.929, 117.585, -2.405]
  MoveL 30 to (13.7, -4.24, -14.7) mm, rotated rx 0 ry 60.72 rz 14.37 deg; joints [-92.707, -109.459, -108.04, -68.314, 118.576, -2.986]
  MoveL 31 to (13.7, -3.22, -14.96) mm, rotated rx 0 ry 59.82 rz 12.18 deg; joints [-93.141, -108.694, -109.698, -65.546, 119.474, -3.527]
  MoveL 32 to (13.7, -2.19, -15.14) mm, rotated rx 0 ry 59.06 rz 9.9 deg; joints [-93.521, -107.926, -111.395, -62.628, 120.269, -4.016]
  MoveL 33 to (13.7, -1.15, -15.26) mm, rotated rx 0 ry 58.47 rz 7.55 deg; joints [-93.841, -107.162, -113.123, -59.565, 120.952, -4.441]
  MoveL 34 to (13.7, -0.1, -15.3) mm, rotated rx 0 ry 58.03 rz 5.13 deg; joints [-94.099, -106.408, -114.875, -56.366, 121.511, -4.79]
  MoveL 35 to (13.7, 0.95, -15.27) mm, rotated rx 0 ry 57.76 rz 2.67 deg; joints [-94.288, -105.669, -116.641, -53.04, 121.935, -5.05]
  MoveL 36 to (13.7, 1.99, -15.17) mm, rotated rx 0 ry 57.67 rz 0.18 deg; joints [-94.406, -104.952, -118.411, -49.602, 122.212, -5.209]
  MoveL 37 to (13.7, 3.03, -15) mm, rotated rx 0 ry 57.74 rz -2.3 deg; joints [-94.446, -104.261, -120.178, -46.07, 122.33, -5.26]
  MoveL 38 to (13.7, 4.05, -14.75) mm, rotated rx 0 ry 57.98 rz -4.77 deg; joints [-94.404, -103.599, -121.931, -42.466, 122.278, -5.193]
  MoveL 39 to (13.7, 5.05, -14.44) mm, rotated rx 0 ry 58.39 rz -7.19 deg; joints [-94.274, -102.97, -123.662, -38.814, 122.045, -5.004]
  MoveL 40 to (13.7, 6.03, -14.06) mm, rotated rx 0 ry 58.97 rz -9.56 deg; joints [-94.051, -102.373, -125.364, -35.142, 121.623, -4.693]
  MoveL 41 to (13.7, 6.98, -13.61) mm, rotated rx 0 ry 59.7 rz -11.85 deg; joints [-93.73, -101.809, -127.028, -31.482, 121.001, -4.26]
  MoveL 42 to (13.7, 7.9, -13.1) mm, rotated rx 0 ry 60.58 rz -14.05 deg; joints [-93.306, -101.276, -128.649, -27.866, 120.174, -3.71]
  MoveL 43 to (13.7, 8.78, -12.53) mm, rotated rx 0 ry 61.6 rz -16.15 deg; joints [-92.773, -100.772, -130.219, -24.327, 119.135, -3.05]
  MoveL 44 to (13.7, 9.62, -11.9) mm, rotated rx 0 ry 62.76 rz -18.13 deg; joints [-92.128, -100.292, -131.734, -20.9, 117.882, -2.288]
  MoveL 45 to (13.7, 10.41, -11.21) mm, rotated rx 0 ry 64.05 rz -19.99 deg; joints [-91.367, -99.832, -133.189, -17.619, 116.415, -1.434]
  MoveL 46 to (13.7, 11.15, -10.47) mm, rotated rx 0 ry 65.45 rz -21.73 deg; joints [-90.486, -99.388, -134.579, -14.513, 114.733, -0.497]
  MoveL 47 to (13.7, 11.84, -9.68) mm, rotated rx 0 ry 66.95 rz -23.33 deg; joints [-89.485, -98.955, -135.901, -11.615, 112.843, 0.513]
  MoveL 48 to (13.7, 12.48, -8.85) mm, rotated rx 0 ry 68.56 rz -24.8 deg; joints [-88.363, -98.53, -137.15, -8.95, 110.75, 1.589]
  MoveL 49 to (13.7, 13.06, -7.97) mm, rotated rx 0 ry 70.25 rz -26.13 deg; joints [-87.123, -98.111, -138.322, -6.543, 108.466, 2.723]
  MoveL 50 to (13.7, 13.57, -7.06) mm, rotated rx 0 ry 72.02 rz -27.33 deg; joints [-85.769, -97.694, -139.411, -4.419, 106.004, 3.91]
  MoveL 51 to (13.7, 14.03, -6.11) mm, rotated rx 0 ry 73.85 rz -28.4 deg; joints [-84.307, -97.28, -140.412, -2.595, 103.38, 5.146]
  MoveL 52 to (13.7, 14.41, -5.14) mm, rotated rx 0 ry 75.75 rz -29.34 deg; joints [-82.748, -96.869, -141.319, -1.091, 100.616, 6.428]
  MoveL 53 to (13.7, 14.73, -4.14) mm, rotated rx 0 ry 77.7 rz -30.14 deg; joints [-81.105, -96.46, -142.126, 0.079, 97.735, 7.755]
  MoveL 54 to (13.7, 14.98, -3.12) mm, rotated rx 0 ry 79.7 rz -30.82 deg; joints [-79.394, -96.058, -142.826, 0.902, 94.763, 9.127]
  MoveL 55 to (13.7, 15.16, -2.08) mm, rotated rx 0 ry 81.73 rz -31.37 deg; joints [-77.633, -95.664, -143.412, 1.367, 91.732, 10.542]
  MoveL 56 to (13.7, 15.26, -1.04) mm, rotated rx 0 ry 83.79 rz -31.79 deg; joints [-75.844, -95.282, -143.877, 1.468, 88.674, 12.001]
  MoveL 57 to (13.7, 15.3, 0.01) mm, rotated rx 0 ry 85.87 rz -32.1 deg; joints [-74.049, -94.915, -144.217, 1.2, 85.622, 13.503]
  MoveL 58 to (13.7, 15.26, 1.06) mm, rotated rx 0 ry 87.96 rz -32.28 deg; joints [-72.272, -94.57, -144.426, 0.563, 82.611, 15.047]
  MoveL 59 to (13.7, 15.15, 2.1) mm, rotated rx -180 ry 89.94 rz 147.67 deg; joints [-70.536, -94.25, -144.498, -0.44, 79.675, 16.629]
  MoveL 60 to (13.7, 14.97, 3.14) mm, rotated rx -180 ry 87.84 rz 147.73 deg; joints [-68.864, -93.962, -144.432, -1.801, 76.846, 18.246]
  MoveL 61 to (13.7, 14.72, 4.15) mm, rotated rx -180 ry 85.74 rz 147.92 deg; joints [-67.276, -93.711, -144.225, -3.506, 74.154, 19.891]
  MoveL 62 to (13.7, 14.4, 5.15) mm, rotated rx -180 ry 83.66 rz 148.23 deg; joints [-65.789, -93.504, -143.876, -5.538, 71.624, 21.554]
  MoveL 63 to (13.7, 14.02, 6.13) mm, rotated rx -180 ry 81.61 rz 148.66 deg; joints [-64.417, -93.348, -143.386, -7.875, 69.278, 23.224]
  MoveL 64 to (13.7, 13.56, 7.08) mm, rotated rx -180 ry 79.58 rz 149.22 deg; joints [-63.171, -93.249, -142.756, -10.489, 67.134, 24.886]
  MoveL 65 to (13.7, 13.05, 7.99) mm, rotated rx 180 ry 77.59 rz 149.9 deg; joints [-62.057, -93.214, -141.99, -13.35, 65.204, 26.525]
  MoveL 66 to (13.7, 12.47, 8.86) mm, rotated rx -180 ry 75.64 rz 150.72 deg; joints [-61.08, -93.251, -141.092, -16.422, 63.497, 28.12]
  MoveL 67 to (13.7, 11.83, 9.7) mm, rotated rx 180 ry 73.74 rz 151.66 deg; joints [-60.241, -93.364, -140.067, -19.67, 62.016, 29.65]
  MoveL 68 to (13.7, 11.14, 10.49) mm, rotated rx -180 ry 71.91 rz 152.73 deg; joints [-59.537, -93.559, -138.923, -23.055, 60.763, 31.094]
  MoveL 69 to (13.7, 10.39, 11.23) mm, rotated rx 180 ry 70.15 rz 153.94 deg; joints [-58.966, -93.838, -137.666, -26.539, 59.733, 32.428]
  MoveL 70 to (13.7, 9.6, 11.91) mm, rotated rx 180 ry 68.46 rz 155.28 deg; joints [-58.522, -94.203, -136.307, -30.085, 58.922, 33.63]
  MoveL 71 to (13.7, 8.76, 12.54) mm, rotated rx -180 ry 66.86 rz 156.76 deg; joints [-58.2, -94.653, -134.853, -33.657, 58.321, 34.679]
  MoveL 72 to (13.7, 7.88, 13.11) mm, rotated rx -180 ry 65.36 rz 158.37 deg; joints [-57.992, -95.187, -133.316, -37.223, 57.92, 35.556]
  MoveL 73 to (13.7, 6.96, 13.62) mm, rotated rx 180 ry 63.97 rz 160.11 deg; joints [-57.892, -95.799, -131.707, -40.755, 57.708, 36.246]
  MoveL 74 to (13.7, 6.01, 14.07) mm, rotated rx -180 ry 62.69 rz 161.98 deg; joints [-57.893, -96.484, -130.035, -44.228, 57.674, 36.736]
  MoveL 75 to (13.7, 5.04, 14.45) mm, rotated rx 180 ry 61.54 rz 163.97 deg; joints [-57.987, -97.235, -128.313, -47.621, 57.806, 37.018]
  MoveL 76 to (13.7, 4.03, 14.76) mm, rotated rx -180 ry 60.52 rz 166.07 deg; joints [-58.167, -98.043, -126.55, -50.918, 58.09, 37.09]
  MoveL 77 to (13.7, 3.01, 15) mm, rotated rx -180 ry 59.65 rz 168.28 deg; joints [-58.427, -98.901, -124.758, -54.105, 58.514, 36.954]
  MoveL 78 to (13.7, 1.98, 15.17) mm, rotated rx -180 ry 58.93 rz 170.57 deg; joints [-58.761, -99.799, -122.946, -57.173, 59.067, 36.616]
  MoveL 79 to (13.7, 0.93, 15.27) mm, rotated rx 180 ry 58.36 rz 172.95 deg; joints [-59.161, -100.73, -121.123, -60.115, 59.738, 36.087]
  MoveL 80 to (13.7, -0.12, 15.3) mm, rotated rx -180 ry 57.96 rz 175.37 deg; joints [-59.623, -101.683, -119.3, -62.928, 60.515, 35.383]
  MoveL 81 to (13.7, -1.17, 15.25) mm, rotated rx -180 ry 57.73 rz 177.84 deg; joints [-60.141, -102.652, -117.483, -65.608, 61.388, 34.521]
  MoveL 82 to (13.7, -2.21, 15.14) mm, rotated rx 180 ry 57.67 rz -179.67 deg; joints [-60.711, -103.629, -115.682, -68.156, 62.349, 33.524]
  MoveL 83 to (13.7, -3.24, 14.95) mm, rotated rx 180 ry 57.78 rz -177.19 deg; joints [-61.327, -104.606, -113.903, -70.57, 63.389, 32.413]
  MoveL 84 to (13.7, -4.26, 14.69) mm, rotated rx -180 ry 58.05 rz -174.73 deg; joints [-61.986, -105.577, -112.154, -72.853, 64.499, 31.211]
  MoveL 85 to (13.7, -5.26, 14.37) mm, rotated rx -180 ry 58.5 rz -172.31 deg; joints [-62.683, -106.537, -110.441, -75.006, 65.673, 29.941]
  MoveL 86 to (13.7, -6.23, 13.97) mm, rotated rx 180 ry 59.1 rz -169.96 deg; joints [-63.415, -107.479, -108.771, -77.031, 66.904, 28.625]
  MoveL 87 to (13.7, -7.17, 13.51) mm, rotated rx 180 ry 59.87 rz -167.69 deg; joints [-64.178, -108.399, -107.15, -78.93, 68.187, 27.283]
  MoveL 88 to (13.7, -8.08, 12.99) mm, rotated rx 180 ry 60.78 rz -165.51 deg; joints [-64.969, -109.292, -105.584, -80.704, 69.516, 25.931]
  MoveL 89 to (13.7, -8.95, 12.41) mm, rotated rx -180 ry 61.83 rz -163.43 deg; joints [-65.786, -110.153, -104.078, -82.356, 70.885, 24.586]
  MoveL 90 to (13.7, -9.78, 11.76) mm, rotated rx 180 ry 63.02 rz -161.47 deg; joints [-66.625, -110.98, -102.637, -83.887, 72.291, 23.26]
  MoveL 91 to (13.7, -10.57, 11.07) mm, rotated rx 180 ry 64.32 rz -159.64 deg; joints [-67.483, -111.768, -101.268, -85.298, 73.73, 21.963]
  MoveL 92 to (13.7, -11.3, 10.32) mm, rotated rx -180 ry 65.75 rz -157.93 deg; joints [-68.359, -112.513, -99.975, -86.59, 75.197, 20.702]
  MoveL 93 to (13.7, -11.98, 9.52) mm, rotated rx -180 ry 67.27 rz -156.36 deg; joints [-69.25, -113.214, -98.763, -87.764, 76.69, 19.482]
  MoveL 94 to (13.7, -12.6, 8.67) mm, rotated rx -180 ry 68.9 rz -154.92 deg; joints [-70.154, -113.866, -97.637, -88.822, 78.205, 18.307]
  MoveL 95 to (13.7, -13.17, 7.79) mm, rotated rx 180 ry 72.16 rz -152.88 deg; joints [-71.755, -114.745, -96.055, -90.151, 81.076, 16.384]
  MoveL 96 to (13.7, -13.47, 7.25) mm, rotated rx -180 ry 77.69 rz -150.13 deg; joints [-74.254, -115.98, -93.946, -91.916, 85.802, 13.648]
  Set speed (1000.0 mm/s)
  MoveL 97 to (13.7, -13.47, 7.25) mm, rotated rx -180 ry 77.69 rz -150.13 deg; joints [-74.254, -115.98, -93.946, -91.916, 85.802, 13.648]
  MoveL 98 to (-71.02, -62.13, 28.57) mm, rotated rx -180 ry 77.69 rz -150.13 deg; joints [-73.617, -117.985, -77.421, -106.475, 86.139, 14.191]

--- program MainProgram (robot UR5) ---
  Hide without_bottom
  Hide Lower_weld_path_dense
  Hide hub_weld
  Show without_top
  Show Top_weld_path_dense
  Smooth(1)
  Call upper_vane
  MoveJ (Home)
  Pause 3.0 s
  Hide Top_weld_path_dense
  Hide without_top
  Show Lower_weld_path_dense
  Show hub_weld
  Show without_bottom
  Smooth(1)
  Call lower_vane
  Smooth(1)
  Call hub
  MoveJ (Home)

